	1044: (* Schleppabstand Filter Time ***********************************************************************)	
		getValue(IDxGrp:= 16#6000,	IDxOffs := 16#13,	LEN := SIZEOF(MaxPosLagFilterTime),	pActValue := ADR(MaxPosLagFilterTime),  pSetValue := ADR(SetMaxPosLagFilterTime) );

	1045: (* Physical unit ***********************************************************************)	
		getValue(IDxGrp:= 16#4000,	IDxOffs := 16#5,	LEN := SIZEOF(PhysicalUnit),	pActValue := ADR(PhysicalUnit),  pSetValue := ADR(PhysicalUnit) );
		IF PhysicalUnit[0] = 176 THEN PhysicalUnit := '°'; END_IF		
		
	1046: (*  Drive type ***********************************************************************)	
		getValue(IDxGrp:= 16#7000,	IDxOffs := 16#3,	LEN := SIZEOF(DriveType),	pActValue := ADR(DriveType),  pSetValue := 0 );
			
	ELSE
		state												:= 1;
	END_CASE

(*********************************************************************************************)
END_METHOD

METHOD PROTECTED seqWrite : BOOL //Return value = TRUE if execution finished 
VAR_IN_OUT
	State							:	INT;
END_VAR
(* Write axis parameter ********************************************************************)
	CASE state OF
	1..99: //Wite application spec parameter 
		seqWrite											:= TRUE;
		
	1001: (* Endlagenlimit pos.beschreiben ********************************************************)
		setValue(IDxGrp:= 16#5000,	IDxOffs := 16#E,	LEN := SIZEOF(SetLimitPos),		pActValue := ADR(LimitPos),		pSetValue := ADR(SetLimitPos));

	1002: (* Endlagenlimit neg.beschreiben ********************************************************)
		setValue(IDxGrp:= 16#5000,	IDxOffs := 16#D,	LEN := SIZEOF(SetLimitNeg),		pActValue := ADR(LimitNeg),		pSetValue := ADR(SetLimitNeg));

	1003: (* Endlagenlimit pos. aktiv ****************************************************************)
		IF NOT (SetLimitPosActive XOR LimitPosActive)
			AND NOT WriteAdsPara.BUSY
		THEN 
			state 											:= state + 1;
		ELSE
			_UINT											:= TO_UINT(SetLimitPosActive);
			LimitPosActive									:= SetLimitPosActive;
			setValue(IDxGrp:= 16#5000,	IDxOffs := 16#C,	LEN := SIZEOF(_UINT),		pActValue := 0,		pSetValue := ADR(_UINT));
		END_IF
		
	1004: (* Endlagenlimit neg.aktiv *****************************************************************)
		IF NOT (SetLimitNegActive XOR LimitNegActive) 
			AND NOT WriteAdsPara.BUSY
		THEN 
			state 											:= state + 1;
		ELSE
			_UINT											:= TO_UINT(SetLimitNegActive);
			LimitNegActive									:= SetLimitNegActive; 
			setValue(IDxGrp:= 16#5000,	IDxOffs := 16#B,	LEN := SIZEOF(_UINT),		pActValue := 0,		pSetValue := ADR(_UINT));
		END_IF

	1005: (* Zielfenster setzen **********************************************************************)
		setValue(IDxGrp:= 16#4000,	IDxOffs := 16#16,	LEN := SIZEOF(SetTargetPosWindow),		pActValue := ADR(TargetPosWindow),		pSetValue := ADR(SetTargetPosWindow));

	1006: (* Positionsfenster setzen *****************************************************************)
		setValue(IDxGrp:= 16#4000,	IDxOffs := 16#10,	LEN := SIZEOF(SetPosRangeWindow),		pActValue := ADR(PosRangeWindow),	pSetValue := ADR(SetPosRangeWindow));
		
	1007: (* Bezugsgeschwindigkeit setzen ********************************************************)
		IF AxisType = 2
		THEN 
			state 											:= state +1;
		ELSE
			setValue(IDxGrp:= 16#7000,	IDxOffs := 16#101,	LEN := SIZEOF(SetDynamicsRefVelocity),pActValue := ADR(DynamicsRefVelocity),	pSetValue := ADR(SetDynamicsRefVelocity));
		END_IF


	1008: (* Max.Geschwindigkeit setzen ************************************************************)
		IF AxisType = 2 
		THEN 
			state 											:= state +1;
		ELSE
			setValue(IDxGrp:= 16#4000,	IDxOffs := 16#27,	LEN := SIZEOF(SetDynamicsMaxVelocity),pActValue := ADR(DynamicsMaxVelocity),	pSetValue := ADR(SetDynamicsMaxVelocity));
		END_IF

	1009: (* G0 Geschwindigkeit setzen ****************************************************************)
		setValue(IDxGrp:= 16#4000,	IDxOffs := 16#A,	LEN := SIZEOF(SetG0Velocity),	pActValue := ADR(G0Velocity),	pSetValue := ADR(SetG0Velocity));

	1010: (* Ref.Geschwindigkeit fast setzen *******************************************************)
		setValue(IDxGrp:= 16#4000,	IDxOffs := 16#6,	LEN := SIZEOF(SetRefVelocityPos),	pActValue := ADR(RefVelocityPos),	pSetValue := ADR(SetRefVelocityPos));

	1011: (* Ref.Geschwindigkeit slow setzen *****************************************************)
		setValue(IDxGrp:= 16#4000,	IDxOffs := 16#7,	LEN := SIZEOF(SetRefVelocityNeg),	pActValue := ADR(RefVelocityNeg),	pSetValue := ADR(SetRefVelocityNeg));

	1012: (* Man.Geschwindigkeit fast setzen ******************************************************)
		setValue(IDxGrp:= 16#4000,	IDxOffs := 16#9,	LEN := SIZEOF(SetManVelocityFast),	pActValue := ADR(ManVelocityFast),	pSetValue := ADR(SetManVelocityFast));
		

	1013: (* Man.Geschwindigkeit slow setzen ******************************************************)
		setValue(IDxGrp:= 16#4000,	IDxOffs := 16#8,	LEN := SIZEOF(SetManVelocitySlow),	pActValue := ADR(ManVelocitySlow),	pSetValue := ADR(SetManVelocitySlow));

	1014: (* Kv setzen **************************************************************************************)
		IF AxisType = 2 
		THEN 
			state 											:= state +1;
		ELSE
			setValue(IDxGrp:= 16#6000,	IDxOffs := 16#102,	LEN := SIZEOF(SetKv),pActValue := ADR(Kv),	pSetValue := ADR(SetKv));
		END_IF

	1015: (* Ruck setzen ***********************************************************************************)
		IF AxisType = 2 
		THEN 
			state 											:= state +1;
		ELSE
			setValue(IDxGrp:= 16#4000,	IDxOffs := 16#103,	LEN := SIZEOF(SetJerk),pActValue := ADR(Jerk),	pSetValue := ADR(SetJerk));
		END_IF

	1016: (* Beschleunigung setzen **********************************************************************)
		IF AxisType = 2 
		THEN 
			state 											:= state +1;
		ELSE
			setValue(IDxGrp:= 16#4000,	IDxOffs := 16#101,	LEN := SIZEOF(SetAcc), pActValue := ADR(Acc),	pSetValue := ADR(SetAcc));
		END_IF
	
	1017: (* Verzoegerung setzen ************************************************************************)
		IF AxisType = 2 
		THEN 
			state 											:= state +1;
		ELSE
			setValue(IDxGrp:= 16#4000,	IDxOffs := 16#102,	LEN := SIZEOF(SetDec), pActValue := ADR(Dec),	pSetValue := ADR(SetDec));
		END_IF
		
	1018: (* Schleppabstand setzen **********************************************************************)
		setValue(IDxGrp:= 16#6000,	IDxOffs := 16#12,	LEN := SIZEOF(SetMaxPosLagValue),	pActValue := ADR(MaxPosLagValue),	pSetValue := ADR(SetMaxPosLagValue));

	1019: (* Reserverd *****************************************************************************)
		// Set scaling replaced by Num and Denum  setValue(IDxGrp:= 16#5000,	IDxOffs := 16#6,	LEN := SIZEOF(SetEncScaling),	pActValue := ADR(EncScaling),	pSetValue := ADR(SetEncScaling));
		state 												:= state +1 ;
		
	1020: (* Positions Offset setzen ****************************************************************)
		setValue(IDxGrp:= 16#5000,	IDxOffs := 16#7,	LEN := SIZEOF(SetPosBias),	pActValue := ADR(PosBias),	pSetValue := ADR(SetPosBias));
		
	1021: (* Referenzposition setzen ***************************************************************)
		IF EncType <> 2  AND EncType <> 5 AND EncType <> 7 AND EncType <> 11  AND EncType <> 12 
		THEN
			setValue(IDxGrp:= 16#5000,	IDxOffs := 16#103,	LEN := SIZEOF(SetCalibrationValue),	pActValue := ADR(CalibrationValue),	pSetValue := ADR(SetCalibrationValue));
		ELSE
			state 											:= state +1 ;
		END_IF

	1022: (* Bremsweg positiv **********************************************************************)
		IF AxisType = 2 
		THEN 
			state 											:= state +1;
		ELSE
			setValue(IDxGrp:= 16#4000,	IDxOffs := 16#303,	LEN := SIZEOF(SetBreakingDistancePos), pActValue := ADR(BreakingDistancePos),	pSetValue := ADR(SetBreakingDistancePos));
		END_IF

	1023: (* Bremsweg negativ *********************************************************************)
		IF AxisType = 2
		THEN 
			state 											:= state +1;
		ELSE
			setValue(IDxGrp:= 16#4000,	IDxOffs := 16#304,	LEN := SIZEOF(SetBreakingDistanceNeg), pActValue := ADR(BreakingDistanceNeg),	pSetValue := ADR(SetBreakingDistanceNeg));
		END_IF

	1024: (* Schleppueberwachung ****************************************************************************)
		IF SetMaxPosLagMonitoring = MaxPosLagMonitoring AND NOT WriteAdsPara.BUSY
		THEN 
			state 											:= state +1;
		ELSE
			_UINT											:= TO_UINT(SetMaxPosLagMonitoring);
			MaxPosLagMonitoring								:= SetMaxPosLagMonitoring;					
			setValue(IDxGrp:= 16#6000,	IDxOffs := 16#10,	LEN := SIZEOF(_UINT),	pActValue := 0,	pSetValue := ADR(_UINT));
		END_IF

	1025: (* Referenzierflag ****************************************************************************)
		IF RefFlag = SetRefFlag AND NOT WriteAdsPara.BUSY
		THEN 
			state 											:= state +1;
		ELSE
			_UINT											:= TO_UINT(SetRefFlag);
			RefFlag											:= SetRefFlag;
			setValue(IDxGrp:= 16#5100,	IDxOffs := 16#9,	LEN := SIZEOF(_UINT), pActValue := 0,	pSetValue := ADR(_UINT));
		END_IF
		
	1026: (* PosfensterAktiv ****************************************************************************)
		IF SetPosRangeWindowMonitoring = PosRangeWindowMonitoring AND NOT WriteAdsPara.BUSY
		THEN 
			state 											:= state +1;
		ELSE
			_UINT											:= TO_UINT(SetPosRangeWindowMonitoring);
			PosRangeWindowMonitoring						:= SetPosRangeWindowMonitoring;
			setValue(IDxGrp:= 16#4000,	IDxOffs := 16#F,	LEN := SIZEOF(_UINT), pActValue := 0,	pSetValue := ADR(_UINT));
		END_IF

	1027: (* ZielfensterAktiv ****************************************************************************)
		IF SetTargetPosWindowMonitoring = TargetPosWindowMonitoring AND NOT WriteAdsPara.BUSY
		THEN 
			state 											:= state +1;
		ELSE
			_UINT											:= TO_UINT(SetTargetPosWindowMonitoring);
			TargetPosWindowMonitoring						:= SetTargetPosWindowMonitoring;
			setValue(IDxGrp:= 16#4000,	IDxOffs := 16#15,	LEN := SIZEOF(_UINT), pActValue := 0,	pSetValue := ADR(_UINT));
		END_IF

	1028: (* Modulofaktor ****************************************************************************)
		setValue(IDxGrp:= 16#5000,	IDxOffs := 16#9,	LEN := SIZEOF(SetModuloFactor), pActValue := ADR(ModuloFactor),	pSetValue := ADR(SetModuloFactor));
		
	1029: (* Enc. Zaehlrichtung ****************************************************************************)
		IF SetInvertEncCoutingDir = InvertEncCoutingDir AND NOT WriteAdsPara.BUSY
		THEN 
			state 											:= state +1;
		ELSE
			_UINT											:= TO_UINT(SetInvertEncCoutingDir);
			InvertEncCoutingDir								:= SetInvertEncCoutingDir;
			setValue(IDxGrp:= 16#5000,	IDxOffs := 16#8,	LEN := SIZEOF(_UINT), pActValue := 0,	pSetValue := ADR(_UINT));
		END_IF

	1030: (* Drive  ****************************************************************************)
		IF SetInvertMotorPolarity = InvertMotorPolarity AND NOT WriteAdsPara.BUSY
		THEN 
			state 											:= state +1;
		ELSE
			_UINT											:= TO_UINT(SetInvertMotorPolarity);
			InvertMotorPolarity								:= SetInvertMotorPolarity;
			setValue(IDxGrp:= 16#7000,	IDxOffs := 16#6,	LEN := SIZEOF(_UINT), pActValue := 0,	pSetValue := ADR(_UINT));
		END_IF
		
		
	1031: (* Enc. Modulo start tolerance ****************************************************************************)
		setValue(IDxGrp:= 16#5000,	IDxOffs := 16#1B,	LEN := SIZEOF(SetToleranceWindowModuloStart), pActValue := ADR(ToleranceWindowModuloStart),	pSetValue := ADR(SetToleranceWindowModuloStart));

	1032: (* Set calibration cam search direction inverted ***************************************************************)
		IF SetCalibrInvertDirForCamSearch = CalibrInvertDirForCamSearch	AND NOT WriteAdsPara.BUSY
			OR_ELSE(EncType = 2  OR EncType = 5 OR EncType = 7 OR EncType = 11  OR EncType = 12)
		THEN 
			state 											:= state +1;
		ELSE
			_UINT											:= TO_UINT(SetCalibrInvertDirForCamSearch);
			CalibrInvertDirForCamSearch						:= SetCalibrInvertDirForCamSearch;
			setValue(IDxGrp:= 16#5000,	IDxOffs := 16#101,	LEN := SIZEOF(_UINT), pActValue := 0,	pSetValue := ADR(_UINT));
		END_IF

	1033: (* Set calibration impuls search direction inverted ***************************************************************)
		IF SetCalibrInvertDirForSyncImpSearch = CalibrInvertDirForSyncImpSearch AND NOT WriteAdsPara.BUSY
			OR_ELSE(EncType = 2  OR EncType = 5 OR EncType = 7 OR EncType = 11  OR EncType = 12)
		THEN 
			state 											:= state +1;
		ELSE
			_UINT											:= TO_UINT(SetCalibrInvertDirForSyncImpSearch);
			CalibrInvertDirForSyncImpSearch					:= SetCalibrInvertDirForSyncImpSearch;
			setValue(IDxGrp:= 16#5000,	IDxOffs := 16#102,	LEN := SIZEOF(_UINT), pActValue := 0,	pSetValue := ADR(_UINT));
		END_IF
		
	1034: (* Set calibration mode ***************************************************************)
		IF SetCalibrationMode = CalibrationMode  AND NOT WriteAdsPara.BUSY
			OR_ELSE(EncType = 2  OR EncType = 5 OR EncType = 7 OR EncType = 11  OR EncType = 12)
		THEN 
			state 											:= state +1;		
		ELSE
			setValue(IDxGrp:= 16#5000,	IDxOffs := 16#107,	LEN := SIZEOF(SetCalibrationMode), pActValue := ADR(CalibrationMode),	pSetValue := ADR(SetCalibrationMode));
		END_IF

	1035: (* Scaling numerator **************************************)
		setValue(IDxGrp:= 16#5000,	IDxOffs := 16#23,	LEN := SIZEOF(SetEncScalingNumerator),	pActValue := ADR(EncScalingNumerator),  pSetValue := ADR(SetEncScalingNumerator) );	
			
	1036: (* Scaling denumerator **************************************)
		setValue(IDxGrp:= 16#5000,	IDxOffs := 16#24,	LEN := SIZEOF(SetEncScalingDenominator),	pActValue := ADR(EncScalingDenominator),  pSetValue := ADR(SetEncScalingDenominator) );
		
		//Calculate Act Scaling 
		IF NOT Error THEN  EncScaling	:= EncScalingNumerator / EncScalingDenominator; END_IF
		
	1037: (* Reference system **************************************)
		setValue(IDxGrp:= 16#5000,	IDxOffs := 16#19,	LEN := SIZEOF(SetReferenceSystem),	pActValue := ADR(ReferenceSystem),  pSetValue := ADR(SetReferenceSystem) );	
	
	1038: (* Schleppueberwachung Zeit ****************************************************************************)
		setValue(IDxGrp:= 16#6000,	IDxOffs := 16#13,	LEN := SIZEOF(SetMaxPosLagFilterTime),	pActValue := ADR(MaxPosLagFilterTime),	pSetValue := ADR(SetMaxPosLagFilterTime));
	
	ELSE
		state 												:= 1 ;
	END_CASE
	
(***********************************************************************************************)
END_METHOD

METHOD PROTECTED setValue : BOOL //Return value = TRUE if execution finished and state incremented 
VAR_INPUT
	IDxGrp						:	UDINT;
	IDxOffs						:	UDINT;
	Len							:	UDINT;
	pActValue					:	PVOID; //Address of variable for actual value, can be zero if no corresponding acual value variable exists
	pSetValue					:	PVOID; //Address of variable for set value variable
END_VAR

IF pActValue <> 0 AND pSetValue <> 0 AND_THEN MEMCMP(pSetValue, pActValue, Len) = 0
THEN //Skip write parameter if set and actual value are equel
	state													:= state + 1;	
	setValue												:= TRUE;
ELSE
	WriteAdsPara( Write := TRUE, IdxGrp :=IDxGrp+AxisId, IdxOffs:=IDxOffs, LEN:=Len, SrcAddr:=pSetValue );
	IF NOT WriteAdsPara.BUSY
	THEN
		IF NOT WriteAdsPara.ERR
		THEN
			IF pActValue <> 0 THEN MEMCPY(pActValue, pSetValue, Len); END_IF	
			state											:= state + 1;
		ELSE
			Busy											:= FALSE;
			Error											:= TRUE;
			ErrorId											:= WriteAdsPara.ERRID;
			ErrorText										:= CONCAT('Error write parameter in state:' , TO_STRING(state * -1));
			ErrorText										:= CONCAT(ErrorText , ' Id:');
			ErrorText										:= CONCAT(ErrorText , TO_STRING(ErrorId));
			State											:= 9999;
		END_IF
		WriteAdsPara (Write := FALSE);
		setValue											:= TRUE;
	END_IF		
END_IF
END_METHOD

END_FUNCTION_BLOCK

// POUs/Motion/TF50xx-NC/00_Base/I_AxNcPTP
INTERFACE I_AxNcPTP EXTENDS I_AxNcBase

{attribute 'monitoring' := 'call'}
PROPERTY rMotion : REFERENCE TO AxMotion
GET
END_GET
END_PROPERTY

END_INTERFACE

// POUs/Motion/TF50xx-NC/01_Main/AxMotion
{attribute 'no_check'}
//Nc-axis motion control - start/stop axis  
//based on Tc2_MC2 library
FUNCTION_BLOCK AxMotion EXTENDS AxFbBase
VAR_OUTPUT CONSTANT
	FNC_HALT												:	INT := 0;
	FNC_STOP												:	INT := 1;
	FNC_MOVE_JOG											:	INT := 2;
	FNC_MOVE_ABS											:	INT := 3;
	FNC_MOVE_REL											:	INT := 4;
	FNC_MOVE_ADD											:	INT := 5;
	FNC_MOVE_MOD											:	INT := 6;
	FNC_MOVE_VELO											:	INT := 7;
END_VAR
VAR_INPUT
	Fnc														:	INT (FNC_HALT..FNC_MOVE_VELO) := FNC_HALT;
	JogFwd													:	BOOL := FALSE;
	JogBwd													:	BOOL	:= FALSE;
	BufferMode												:	MC_BufferMode := MC_Aborting;(* 	MC_Aborting,
																											MC_Buffered,
																											MC_BlendingLow,
																											MC_BlendingPrevious,
																											MC_BlendingNext,
																											MC_BlendingHigh *)
	Direction												:	MC_Direction := MC_POSITIVE_DIRECTION;	(*	MC_POSITIVE_DIRECTION,
																														   MC_SHORTeSTATE.WAY,
																														   MC_NEGATIVE_DIRECTION,
																														   MC_CURRENT_DIRECTION *)
	JogMode													:	E_JogMode := MC_JOGMODE_STANDARD_SLOW;	(*	MC_JOGMODE_STANDARD_SLOW
																															MC_JOGMODE_STANDARD_FAST
																															MC_JOGMODE_CONTINOUS
																															MC_JOGMODE_INCHING 
																															MC_JOGeMODE.INCHING_MODULO *)
	Target													:	LREAL; (* Zielposition *)
	Velo														: 	LREAL; (* Zielgeschwindigkeit *)
	Jerk														:	LREAL := 0.0 ; (* Bei 0 werden wird der Ruck aus dem TCManager uebernommen *)
	Acc														:	LREAL := 0.0; (* Bei 0 werden wird die Beschleunigung aus dem TCManager uebernommen *)
	Dec														:	LREAL := 0.0; (* Bei 0 werden wird die Verzoegerung aus dem TCManager uebernommen *)
	MoveOptions												:	ST_MoveOptions;
END_VAR                     								
VAR_IN_OUT                  								
END_VAR                     								
VAR_OUTPUT                  								
END_VAR
VAR
(* Zwischenspeicher **************************************************************************)
	MemFnc													:	INT := -1;
	MemFncAct												:	INT := -1;
	MCFctTxt												:	STRING(25);
	TrigID													:	INT := 2; (* um mit Trig 1 zu starten *)
	MemBufferMode											:	MC_BufferMode;
	ActSetTarget											:	LREAL;
	ActSetVelo												:	LREAL;
	BusyIntern												:	BOOL;

(* Timer *)

(* Trigger *)
	rtExecuteMethod											:	R_TRIG;

(* Instanzierung der MC Bausteine *******************************************************)
	MC_Halt													: 	MC_Halt;
	MC_Stop													: 	MC_Stop;
	MC_MoveVeloPreTrig										: 	MC_MoveVelocity;
	MC_Jog													: 	MC_Jog;

(* Durch entfernen der Kommentarsymbole koennen noch weitere benötigte MC_Move Varianten
	mit ins Programm genommen werden 
*)
	MC_MoveAbsolute											: 	ARRAY[1..2] OF MC_MoveAbsolute;
	MC_MoveModulo											: 	ARRAY[1..2] OF MC_MoveModulo;
	MC_MoveRelative											: 	ARRAY[1..2] OF MC_MoveRelative;
	MC_MoveAdditive											: 	ARRAY[1..2] OF MC_MoveAdditive; 
	MC_MoveVelocity											: 	ARRAY[1..2] OF MC_MoveVelocity; 

(* Dummy Speicher **********************************************************)
	i														: INT := 0 ;

(* Skalierungsfaktor ermitteln *********************************************
	Skalierungsfaktor von 0.1 eintragen. Istpositon "Anfang" merken.
	Antrieb um einen realen Wert "X" mm verfahren. Differenz der
	momentanen Istposition zur Istposition "Anfang" ermitteln.
	SKalierungsfaktor =		realer Fahrweg 
							---------------------------
							Differenz der Istpositionen
*)
END_VAR

	(* Axis motion control 													*)
	(************************************************************************)

(* Execute ***************************************************************************************)
	rtExecute(CLK := Execute XOR(JogBwd AND NOT JogFwd OR JogFwd AND NOT JogBwd));	
	IF rtExecute.Q AND NOT rtExecuteMethod.Q
	THEN
		MemFnc 												:= SEL(JogBwd OR JogFwd, Fnc, FNC_MOVE_JOG) ;
		Busy												:= TRUE;
		Done												:= FALSE;
		Active												:= FALSE;
		Error												:= FALSE;
		ErrorID												:= 0;
		CmdAborted											:= FALSE;
		ErrorText											:= '';
	END_IF

(* Call Method ***********************************************************************************)
	CASE MemFnc OF
	FNC_STOP												:	Stop(Execute);
	FNC_HALT												:	Halt(Execute);
	FNC_MOVE_JOG											:	MoveJog(Execute);
	FNC_MOVE_ABS											:	MoveAbs(Execute);
	FNC_MOVE_REL											:	MoveRel(Execute);
	FNC_MOVE_ADD											:	MoveAdd(Execute);
	FNC_MOVE_MOD											:	MoveMod(Execute);
	FNC_MOVE_VELO											:	MoveVelo(Execute);
	-1:
		IF NOT rtExecute.CLK
		THEN
			Busy											:= FALSE;
			Done											:= FALSE;
			Error											:= FALSE;
			ErrorID											:= 0;
			Active											:= FALSE;
			CmdAborted										:= FALSE;
			ErrorText										:= '';
		END_IF
	ELSE
		Busy												:= FALSE;
		Done												:= FALSE;
		Active												:= FALSE;
		Error												:= Execute;
		ErrorID												:= E_AdsErr.DEVICE_INVALIDPARM;
		CmdAborted											:= FALSE;
		ErrorText											:= CONCAT('invalid parameter value(s) Fnc no: ' , INT_TO_STRING(MemFnc));
	END_CASE

(*************************************************************************************************)

METHOD PRIVATE _MCIntern : BOOL
VAR_INPUT
END_VAR
(* Internal MC Action											*)
(****************************************************************)

(* Check Pointer **********************************************************************)
IF NOT __ISVALIDREF(rAxis) 
THEN
	Busy													:= NOT Error;
	Error													:= TRUE;
	ErrorId													:= E_AdsErr.DEVICE_INVALIDPARM;
	CmdAborted												:= FALSE;
	Done													:= FALSE;
	Active													:= FALSE;
	ErrorText												:= 'Reference rAxis invalid (0)';
	MemFnc													:= SEL(Execute , -1 ,MemFnc); 
	RETURN;
END_IF

(* flag Execute ***********************************************************************)
	rtExecuteMethod(CLK := Execute OR rtExecute.Q);
	IF rtExecuteMethod.Q 
	THEN
		MC_Stop.Execute										:= FALSE;
		MC_Halt.Execute										:= FALSE;
		MC_MoveVeloPreTrig.Execute							:= FALSE;
		MC_MoveModulo[1].Execute 							:= MC_MoveModulo[2].Execute	:= FALSE;
		MC_MoveAbsolute[1].Execute							:= MC_MoveAbsolute[2].Execute	:= FALSE;
		MC_MoveRelative[1].Execute 							:= MC_MoveRelative[2].Execute := FALSE; 
		MC_MoveAdditive[1].Execute 							:= MC_MoveAdditive[2].Execute := FALSE; 
		MC_MoveVelocity[1].Execute 							:= MC_MoveVelocity[2].Execute := FALSE; 
		BusyIntern											:= FALSE;
		MemFncAct 											:= MemFnc;
	END_IF

(* ctrl programm ******************************************************************************)
	CASE MemFncAct OF
	-1: ; //No Fnc started
	FNC_STOP:
		MC_Stop.Execute										:=	Execute; (* Achse Locked solange Stop noch ansteht *)
		MC_Stop.Deceleration 								:= Dec;
		MC_Stop.Jerk 										:= Jerk;
		MC_Stop.Options 									:= MoveOptions;

	FNC_HALT:
		MC_Halt.Execute										:=	NOT MC_Stop.Busy AND Execute; (* Execute if axis is not locked *)
		MC_Halt.BufferMode									:= BufferMode;
		MC_Halt.Deceleration 								:= Dec;
		MC_Halt.Jerk 										:= Jerk;
		MC_Halt.Options 									:= MoveOptions;
		BusyIntern											:= MC_Stop.Busy;

	FNC_MOVE_JOG:
		IF(Execute OR JogBwd OR JogFwd OR MC_Halt.Busy) (* new cmd or stop last cmd busy *)
			AND NOT rAxis.NcToPlc.StateDWord.2  (* NotMoving *)
			AND NOT MC_Jog.Busy (* not if Mc_Jog running *)
			AND NOT rAxis.NcToPlc.StateDWord.5 (* Protected *) (* not if axis coupled or in NCI group *)
			AND NOT MC_Halt.Error AND NOT MC_Halt.CommandAborted
		THEN
			MC_Halt.Execute									:=	TRUE;
			MC_Halt.BufferMode								:= MC_Aborting;
			MC_Halt.Deceleration 							:= Dec;
			MC_Halt.Jerk 									:= Jerk;
			MC_Halt.Options 								:= MoveOptions;
			BusyIntern										:= TRUE;
		ELSE
			MC_Jog.JogBackwards								:= NOT MC_Stop.Busy AND (JogBwd XOR Execute AND Direction = MC_NEGATIVE_DIRECTION);
			MC_Jog.JogForward								:= NOT MC_Stop.Busy AND (JogFwd XOR Execute AND Direction = MC_POSITIVE_DIRECTION);
			MC_Jog.Mode										:= JogMode;
			MC_Jog.Position 								:= Target;
			MC_Jog.Velocity 								:= Velo;
			MC_Jog.Acceleration 							:= Acc;
			MC_Jog.Deceleration 							:= Dec;
			MC_Jog.Jerk 									:= Jerk;
			MC_Halt.Execute									:=	FALSE;
			BusyIntern										:= MC_Stop.Busy;
		END_IF

	FNC_MOVE_ABS..FNC_MOVE_VELO:
		IF MC_Stop.Busy
			OR rAxis.NcToPlc.StateDWord.29 (* MotionCommandsLocked *)
		//	OR MC_Jog.Busy Allow new command even jog is still active
		THEN (* Solange hier rein bis Achse wieder frei und Stop nicht mehr Busy *)
			BusyIntern										:= TRUE;

		ELSIF rAxis.NcToPlc.StateDWord.24 (* CmdBuffered *) 
		THEN (* this section is for aborting a buffered running axis *)
			IF NOT MC_MoveVeloPreTrig.Execute
				AND BufferMode = MC_Aborting
				AND(
				rtExecuteMethod.Q (* new cmd with MC_Aborting to break up current and buffered cmd *)
				OR 		(* or break up current and buffered cmd with new targetpos. *)
				Execute
				AND (Busy OR Done OR CmdAborted) (* dont restart if error is active *)
				AND (ActSetTarget <> Target))
			THEN
				TrigID 										:= 0;
				MC_MoveVeloPreTrig.Execute 					:= TRUE;
				MC_MoveVeloPreTrig.BufferMode 				:= MC_Aborting;
				MC_MoveVeloPreTrig.Velocity 				:= Velo;
				IF rAxis.NcToPlc.StateDWord.10 (* NegativeDirection *) 
				THEN
					MC_MoveVeloPreTrig.Direction 			:= MC_NEGATIVE_DIRECTION;
				ELSE
					MC_MoveVeloPreTrig.Direction 			:= MC_POSITIVE_DIRECTION;
				END_IF
				BusyIntern									:= TRUE;
			ELSE
				;
			END_IF

		ELSE (* ready for start/restart (MC_MoveVeloPreTrig is active) *)
			IF rtExecuteMethod.Q (* new cmd *)
				OR TrigID = 0 (* new cmd with Buffermode aborted *)
				OR(	Execute
				AND (Busy OR Done OR CmdAborted) (* dont restart if error is active *)
				AND (ActSetTarget <> Target OR ActSetVelo <> Velo AND BufferMode = MC_Aborting)) (* restart only with new velo if bufferMode = Aborting *)
			THEN (* new cmd *)
				(* Cancel MoveVeloPreTrig block *)
				IF TrigID = 0 THEN
					MemBufferMode 							:= MC_Aborting;
				ELSE
					MemBufferMode						 	:= BufferMode;
				END_IF

				(* change TrigID *)
				IF TrigID <> 1 THEN
					TrigID 									:= 1;
				ELSE
					TrigID 									:= 2;
				END_IF

				(* Save Act. target and velo *)
				ActSetTarget 								:= Target;
				ActSetVelo 									:= Velo;

				(* Init MC-Blocks *)
				MC_MoveModulo[1].Execute 					:= MC_MoveModulo[2].Execute	:= FALSE;
				MC_MoveAbsolute[1].Execute					:= MC_MoveAbsolute[2].Execute	:= FALSE;
				MC_MoveRelative[1].Execute 					:= MC_MoveRelative[2].Execute := FALSE; 
				MC_MoveAdditive[1].Execute 					:= MC_MoveAdditive[2].Execute := FALSE; 
				MC_MoveVelocity[1].Execute 					:= MC_MoveVelocity[2].Execute := FALSE; 
			END_IF

			CASE MemFncAct OF
			FNC_MOVE_ABS:(* Absolute *);
				MC_MoveAbsolute[TrigID].Execute				:= Execute OR BusyIntern;
				MC_MoveAbsolute[TrigID].BufferMode 			:= MemBufferMode;
				MC_MoveAbsolute[TrigID].Position 			:= Target;
				MC_MoveAbsolute[TrigID].Velocity 			:= Velo;
				MC_MoveAbsolute[TrigID].Acceleration 		:= Acc;
				MC_MoveAbsolute[TrigID].Deceleration 		:= Dec;
				MC_MoveAbsolute[TrigID].Jerk 				:= Jerk;
				MC_MoveAbsolute[TrigID].Options 			:= MoveOptions;

			FNC_MOVE_MOD:(* Modulo *);
				MC_MoveModulo[TrigID].Execute				:= Execute OR BusyIntern;
				MC_MoveModulo[TrigID].BufferMode 			:= MemBufferMode;
				MC_MoveModulo[TrigID].Position 				:= Target;
				MC_MoveModulo[TrigID].Direction 			:= Direction;
				MC_MoveModulo[TrigID].Velocity 				:= Velo;
				MC_MoveModulo[TrigID].Acceleration 			:= Acc;
				MC_MoveModulo[TrigID].Deceleration 			:= Dec;
				MC_MoveModulo[TrigID].Jerk 					:= Jerk;
				MC_MoveModulo[TrigID].Options 				:= MoveOptions;
			
			FNC_MOVE_REL: (* Relativ *)
				MC_MoveRelative[TrigID].Execute				:= Execute OR BusyIntern;
				MC_MoveRelative[TrigID].BufferMode 			:= MemBufferMode;
				MC_MoveRelative[TrigID].Distance 			:= Target;
				MC_MoveRelative[TrigID].Velocity 			:= Velo;
				MC_MoveRelative[TrigID].Acceleration 		:= Acc;
				MC_MoveRelative[TrigID].Deceleration	 	:= Dec;
				MC_MoveRelative[TrigID].Jerk 				:= Jerk;
				MC_MoveRelative[TrigID].Options 			:= MoveOptions;
		
			FNC_MOVE_ADD:(* Rel.Additive *);
				MC_MoveAdditive[TrigID].Execute				:= Execute OR BusyIntern;
				MC_MoveAdditive[TrigID].BufferMode 			:= MemBufferMode;
				MC_MoveAdditive[TrigID].Distance 			:= Target;
				MC_MoveAdditive[TrigID].Velocity 			:= Velo;
				MC_MoveAdditive[TrigID].Acceleration	 	:= Acc;
				MC_MoveAdditive[TrigID].Deceleration	 	:= Dec;
				MC_MoveAdditive[TrigID].Jerk 				:= Jerk;
				MC_MoveAdditive[TrigID].Options 			:= MoveOptions;
			
			FNC_MOVE_VELO:(* Velocity *);
				MC_MoveVelocity[TrigID].Execute				:= Execute OR BusyIntern;
				MC_MoveVelocity[TrigID].BufferMode 			:= MemBufferMode;
				MC_MoveVelocity[TrigID].Direction 			:= Direction;
				MC_MoveVelocity[TrigID].Velocity 			:= Velo;
				MC_MoveVelocity[TrigID].Acceleration 		:= Acc;
				MC_MoveVelocity[TrigID].Deceleration 		:= Dec;
				MC_MoveVelocity[TrigID].Jerk 				:= Jerk;
				MC_MoveVelocity[TrigID].Options 			:= MoveOptions;
			
			ELSE
				MC_Halt.Execute								:=	TRUE; // axis locked as long as Stop is set 
				Error										:= TRUE;
				ErrorId										:= E_AdsErr.DEVICE_INVALIDPARM;
				ErrorText									:= CONCAT('invalid parameter value(s) - Fnc no ', INT_TO_STRING(MemFncAct)) ;
			END_CASE

			(* Reset busy intern *)
			MC_MoveVeloPreTrig.Execute 						:= FALSE;
			BusyIntern										:= FALSE;
		END_IF
	ELSE
		MC_Halt.Execute										:=	TRUE; // axis locked as long as Stop is set
		Error												:= TRUE;
		ErrorId												:= E_AdsErr.DEVICE_INVALIDPARM;
		ErrorText											:= CONCAT('invalid parameter value(s) - Fnc no ', INT_TO_STRING(MemFncAct)) ;
	END_CASE

(****************************************************************************)
(* Work MC Blocks 															*)
(****************************************************************************)

	(* Halt/Stop *)
	MC_Stop(Axis	:= rAxis);
	MC_Halt(Axis	:= rAxis);

	(* Jog *)
	IF MC_Jog.JogBackwards OR MC_Jog.JogForward OR MC_Jog.Busy
		OR MC_Jog.Done OR MC_Jog.Active
		OR MC_Jog.CommandAborted OR MC_Jog.Error
	THEN
		MC_Jog( Axis :=	rAxis);
		MC_Jog.JogBackwards									:= FALSE;
		MC_Jog.JogForward									:= FALSE;
	END_IF

	(* Positionierungen ********************************************)
	(* MC Move Velo PreTrig 1 *)
	IF MC_MoveVeloPreTrig.Execute OR MC_MoveVeloPreTrig.Busy
		OR MC_MoveVeloPreTrig.InVelocity OR MC_MoveVeloPreTrig.Active
		OR MC_MoveVeloPreTrig.CommandAborted OR MC_MoveVeloPreTrig.Error
	THEN
		MC_MoveVeloPreTrig(Axis	:=	rAxis);
	END_IF

	(* Run MC *)
	IF MC_MoveAbsolute[1].Execute OR MC_MoveAbsolute[1].Busy
		OR MC_MoveAbsolute[1].Done OR MC_MoveAbsolute[1].Active
		OR MC_MoveAbsolute[1].CommandAborted OR MC_MoveAbsolute[1].Error
	THEN
		MC_MoveAbsolute[1]( Axis	:=	rAxis);
	END_IF

	IF MC_MoveModulo[1].Execute OR MC_MoveModulo[1].Busy
		OR MC_MoveModulo[1].Done OR MC_MoveModulo[1].Active
		OR MC_MoveModulo[1].CommandAborted OR MC_MoveModulo[1].Error
	THEN
		MC_MoveModulo[1](Axis	:=	rAxis);
	END_IF
	
	IF MC_MoveRelative[1].Execute OR MC_MoveRelative[1].Busy
		OR MC_MoveRelative[1].Done OR MC_MoveRelative[1].Active
		OR MC_MoveRelative[1].CommandAborted OR MC_MoveRelative[1].Error
	THEN
		MC_MoveRelative[1](Axis	:=	rAxis);
	END_IF
	
	IF MC_MoveAdditive[1].Execute OR MC_MoveAdditive[1].Busy
		OR MC_MoveAdditive[1].Done OR MC_MoveAdditive[1].Active
		OR MC_MoveAdditive[1].CommandAborted OR MC_MoveAdditive[1].Error
	THEN
		MC_MoveAdditive[1](Axis	:=	rAxis);
	END_IF
	
	IF MC_MoveVelocity[1].Execute OR MC_MoveVelocity[1].Busy
		OR MC_MoveVelocity[1].Active OR MC_MoveVelocity[1].InVelocity
		OR MC_MoveVelocity[1].CommandAborted OR MC_MoveVelocity[1].Error
	THEN
		MC_MoveVelocity[1](Axis	:=	rAxis);
	END_IF

	(* MC Move Velo PreTrig 2 **************************************)
	(* Run Trig 2 *)
	IF MC_MoveAbsolute[2].Execute OR MC_MoveAbsolute[2].Busy
		OR MC_MoveAbsolute[2].Done OR MC_MoveAbsolute[2].Active
		OR MC_MoveAbsolute[2].CommandAborted OR MC_MoveAbsolute[2].Error
	THEN
		MC_MoveAbsolute[2](Axis	:=	rAxis);
	END_IF

	IF MC_MoveModulo[2].Execute OR MC_MoveModulo[2].Busy
		OR MC_MoveModulo[2].Done OR MC_MoveModulo[2].Active
		OR MC_MoveModulo[2].CommandAborted OR MC_MoveModulo[2].Error
	THEN
		MC_MoveModulo[2](Axis	:=	rAxis);
	END_IF

	
	IF MC_MoveRelative[2].Execute OR MC_MoveRelative[2].Busy
		OR MC_MoveRelative[2].Done OR MC_MoveRelative[2].Active
		OR MC_MoveRelative[2].CommandAborted OR MC_MoveRelative[2].Error
	THEN
		MC_MoveRelative[2](Axis	:=	rAxis);
	END_IF
	
	IF MC_MoveAdditive[2].Execute OR MC_MoveAdditive[2].Busy
		OR MC_MoveAdditive[2].Done OR MC_MoveAdditive[2].Active
		OR MC_MoveAdditive[2].CommandAborted OR MC_MoveAdditive[2].Error
	THEN
		MC_MoveAdditive[2](Axis	:=	rAxis);
	END_IF

	
	IF MC_MoveVelocity[2].Execute OR MC_MoveVelocity[2].Busy
		OR MC_MoveVelocity[2].Active OR MC_MoveVelocity[2].InVelocity
		OR MC_MoveVelocity[2].CommandAborted OR MC_MoveVelocity[2].Error
	THEN
		MC_MoveVelocity[2](Axis	:=	rAxis);
	END_IF

(******************************************************************************)
(* Ctrl Status 																					*)
(******************************************************************************)
	IF MemFncAct = FNC_STOP
	THEN (* as long as MC_Stop running the axis is locked *)
		MCFctTxt											:= 'MC_STOP';
		Done 												:= MC_Stop.Done;
		Busy 												:= MC_Stop.Busy;
		Active 												:= MC_Stop.Active;
		CmdAborted 											:= MC_Stop.CommandAborted;
		Error												:= MC_Stop.Error;
		ErrorId												:= MC_Stop.ErrorId;
		ErrorText											:= SEL(Error , '' ,  CONCAT('Error MC_STOP id: ',  UDINT_TO_STRING(Errorid)));

	ELSIF MemFncAct = FNC_HALT
	THEN
		MCFctTxt											:= 'MC_HALT';
		Done 												:= MC_Halt.Done;
		Busy 												:= MC_Halt.Busy;
		Active 												:= MC_Halt.Active;
		CmdAborted 	 										:= MC_Halt.CommandAborted;
		Error												:= MC_Halt.Error;
		ErrorId												:= MC_Halt.ErrorId;
		ErrorText											:= SEL(Error , '' ,  CONCAT('Error MC_HALT id: ',  UDINT_TO_STRING(Errorid)));

	ELSIF BusyIntern
	THEN
		MCFctTxt											:= CONCAT('BUSY INTERN at Fnc no: ', INT_TO_STRING(MemFncAct));
		Busy												:= BusyIntern;
		Done 												:= FALSE;
		Active 												:= FALSE;
		CmdAborted 											:= FALSE;
		Error												:=	FALSE;
		ErrorId												:= 0;
		ErrorText											:= '';

	ELSIF MemFncAct = FNC_MOVE_JOG
	THEN
		MCFctTxt											:= 'MC_JOG';
		Done 												:= MC_Jog.Done;
		Busy 												:= MC_Jog.Busy;
		Active 												:= MC_Jog.Active;
		CmdAborted 	 										:= MC_Jog.CommandAborted AND NOT rAxis.NcToPlc.StateDWord.26 AND NOT rAxis.NcToPlc.StateDWord.27  (* Software limit exceeded *) ;
		Error												:= MC_Jog.Error;
		ErrorId												:= MC_Jog.ErrorId;
		ErrorText											:= SEL(Error , '' ,  CONCAT('Error MC_JOG id: ',  UDINT_TO_STRING(Errorid)));

	ELSIF MC_MoveVeloPreTrig.Execute
		OR TrigID = 0
	THEN (* Pretrig Block *)
		MCFctTxt											:= 'MC_MoveVeloPreTrig';
		Done												:= FALSE;
		Busy												:= MC_MoveVeloPreTrig.Busy;
		Active 												:= MC_MoveVeloPreTrig.Active;
		CmdAborted 	 										:= MC_MoveVeloPreTrig.CommandAborted;
		Error												:= MC_MoveVeloPreTrig.Error;
		ErrorId												:= MC_MoveVeloPreTrig.ErrorId;
		ErrorText											:= SEL(Error , '' ,  CONCAT('Error MC_MoveVeloPreTrig id: ',  UDINT_TO_STRING(Errorid)));

	ELSIF MemFncAct = FNC_MOVE_ABS
	THEN (* Absolut *)
		MCFctTxt											:= CONCAT('MC_MoveAbs TrigID No:',INT_TO_STRING(TrigID));
		Done 												:= MC_MoveAbsolute[TrigID].Done;
		Busy 												:= MC_MoveAbsolute[TrigID].Busy;
		Active 												:= MC_MoveAbsolute[TrigID].Active;
		CmdAborted 	 										:= MC_MoveAbsolute[TrigID].CommandAborted;
		Error												:= MC_MoveAbsolute[TrigID].Error;
		ErrorId												:= MC_MoveAbsolute[TrigID].ErrorId;
		ErrorText											:= SEL(Error , '' ,  CONCAT('Error MC_MoveAbsolute id: ',  UDINT_TO_STRING(Errorid)));
	
	ELSIF MemFncAct = FNC_MOVE_MOD
	THEN (* Modulo *)
		MCFctTxt											:= CONCAT('MC_MoveModulo TrigID No:',INT_TO_STRING(TrigID));
		Done 												:= MC_MoveModulo[TrigID].Done;
		Busy 												:= MC_MoveModulo[TrigID].Busy;
		Active 												:= MC_MoveModulo[TrigID].Active;
		CmdAborted 											:= MC_MoveModulo[TrigID].CommandAborted;
		Error												:= MC_MoveModulo[TrigID].Error;
		ErrorId												:= MC_MoveModulo[TrigID].ErrorId;
		ErrorText											:= SEL(Error , '' ,  CONCAT('Error MC_MoveModulo id: ',  UDINT_TO_STRING(Errorid)));

	ELSIF MemFncAct = FNC_MOVE_REL
	THEN (* Relativ *)
		MCFctTxt											:= CONCAT('MC_MoveRelative TrigID No:',INT_TO_STRING(TrigID));
		Done 												:= MC_MoveRelative[TrigID].Done;
		Busy 												:= MC_MoveRelative[TrigID].Busy;
		Active 												:= MC_MoveRelative[TrigID].Active;
		CmdAborted 	 										:= MC_MoveRelative[TrigID].CommandAborted;
		Error												:= MC_MoveRelative[TrigID].Error;
		ErrorId												:= MC_MoveRelative[TrigID].ErrorId;
		ErrorText											:= SEL(Error , '' ,  CONCAT('Error MC_MoveRelative id: ',  UDINT_TO_STRING(Errorid)));

	ELSIF MemFncAct = FNC_MOVE_ADD
	THEN (* Rel.Additive *)
		MCFctTxt											:= CONCAT('MC_MoveAdditive TrigID No:',INT_TO_STRING(TrigID));
		Done 												:= MC_MoveAdditive[TrigID].Done;
		Busy 												:= MC_MoveAdditive[TrigID].Busy;
		Active 												:= MC_MoveAdditive[TrigID].Active;
		CmdAborted 	 										:= MC_MoveAdditive[TrigID].CommandAborted;
		Error												:= MC_MoveAdditive[TrigID].Error;
		ErrorId												:= MC_MoveAdditive[TrigID].ErrorId;
		ErrorText											:= SEL(Error , '' ,  CONCAT('Error MC_MoveAdditive id: ',  UDINT_TO_STRING(Errorid)));
		
	ELSIF MemFncAct = FNC_MOVE_VELO
	THEN (* Velocity *)
		MCFctTxt											:= CONCAT('MC_MoveVelo TrigID No:',INT_TO_STRING(TrigID));
		Active 												:= MC_MoveVelocity[TrigID].Active;
		Busy 												:= MC_MoveVelocity[TrigID].Busy ;
		CmdAborted 	 										:= MC_MoveVelocity[TrigID].CommandAborted;
		Error												:= MC_MoveVelocity[TrigID].Error;
		ErrorId												:= MC_MoveVelocity[TrigID].ErrorId;
		ErrorText											:= SEL(Error , '' ,  CONCAT('Error MC_MoveVelocity id: ',  UDINT_TO_STRING(Errorid)));
		
	ELSIF MemFncAct > 0
	THEN
		MCFctTxt											:= CONCAT('Unknown Fnc no:', INT_TO_STRING(MemFncAct));
	ELSE                    							
		MCFctTxt											:= SEL(BusyIntern, 'NoAction' , 'Busy intern');
		Busy												:= BusyIntern;
		Done 												:= FALSE;
		Active 												:= FALSE;
		CmdAborted 											:= FALSE;
		IF Error THEN LastErrorId := ErrorId; END_IF
		Error												:=	FALSE;
		ErrorId												:= 0;
		ErrorText											:= '';
	END_IF

(* End funcktion *********************************************************************************)
	IF 	NOT rtExecuteMethod.CLK 
		AND NOT Busy 
		AND NOT Error 
		AND NOT Done 
		AND NOT Active 
		AND NOT CmdAborted
	THEN																	
		IF MC_Jog.Busy
			OR MC_Halt.Busy
			OR MC_Stop.Busy
			OR MC_MoveVeloPreTrig.Busy
			OR MC_MoveAbsolute[1].Busy OR MC_MoveAbsolute[2].Busy
			OR MC_MoveModulo[1].Busy OR MC_MoveModulo[2].Busy
			OR MC_MoveRelative[1].Busy OR MC_MoveRelative[2].Busy 
			OR MC_MoveAdditive[1].Busy OR MC_MoveAdditive[2].Busy 
			OR MC_MoveVelocity[1].Busy OR MC_MoveVelocity[2].Busy 
		THEN (* Ablauffehler , es darf kein Baustein an dieser Stelle Busy sein *)
			MemFnc											:= -2;
		ELSE                								
			MemFnc											:= -1;
		END_IF              	
	END_IF
	
(* Return value ***********************************************************************************)
	_MCIntern												:= TRUE;

(**************************************************************************************************)
END_METHOD

METHOD PUBLIC halt : BOOL //Return value = TRUE if busy
//required parameter
//rAxis
//BufferMode
//Dec
//Jerk
//MoveOptions
VAR_INPUT
	Execute													:	BOOL;
END_VAR
MemFnc 														:= FNC_HALT;
THIS^.Execute												:= Execute;
_MCIntern();            									
Halt														:= Busy;
END_METHOD

METHOD PUBLIC jogOff : BOOL //Return value = TRUE if executio finished
VAR_INPUT
END_VAR
JogBwd 														:= JogFwd := FALSE;
IF __ISVALIDREF(rAxis)
THEN
	JogOff 													:= MemFnc = FNC_MOVE_JOG AND NOT rAxis.Status.Moving;
ELSE
	JogOff 													:= MemFnc = FNC_MOVE_JOG;
END_IF
END_METHOD

METHOD PUBLIC moveAbs : BOOL //Return value = TRUE if busy
//required parameter
//rAxis
//BufferMode
//Target
//Velo
//Acc
//Dec
//Jerk
//MoveOptions
VAR_INPUT
	Execute													:	BOOL;
END_VAR
MemFnc 														:= FNC_MOVE_ABS;
THIS^.Execute												:= Execute;
_MCIntern();            									
MoveAbs														:= Busy;
END_METHOD

METHOD PUBLIC moveAdd : BOOL //Return value = TRUE if busy
//required parameter
//rAxis
//BufferMode
//Target
//Velo
//Acc
//Dec
//Jerk
//MoveOptions
VAR_INPUT
	Execute													:	BOOL;
END_VAR
MemFnc 														:= FNC_MOVE_ADD;
THIS^.Execute												:= Execute;
_MCIntern();            									
MoveAdd														:= Busy;
END_METHOD

METHOD PUBLIC moveJog : BOOL  //Return value = TRUE if busy
//required parameter
//rAxis
//Direction
//JogMode	
//Target
//Velo
//Acc
//Dec
//Jerk
VAR_INPUT
	Execute													:	BOOL;
END_VAR
MemFnc 														:= FNC_MOVE_JOG;
THIS^.Execute												:= Execute;
_MCIntern();        										
MoveJog														:= Busy;
END_METHOD

METHOD PUBLIC moveMod : BOOL //Return value = TRUE if busy
//required parameter
//rAxis
//BufferMode
//Target
//Direction
//Velo
//Acc
//Dec
//Jerk
//MoveOptions
VAR_INPUT
	Execute													:	BOOL;
END_VAR
MemFnc 														:= FNC_MOVE_MOD;
THIS^.Execute												:= Execute;
_MCIntern();            									
MoveMod														:= Busy;
END_METHOD

METHOD moveRel : BOOL //Return value = TRUE if busy
//required parameter
//rAxis
//BufferMode
//Target
//Velo
//Acc
//Dec
//Jerk
//MoveOptions
VAR_INPUT
	Execute													:	BOOL;
END_VAR
MemFnc 														:= FNC_MOVE_REL;
THIS^.Execute												:= Execute;
_MCIntern();            									
MoveRel														:= Busy;
END_METHOD

METHOD PUBLIC moveVelo : BOOL //Return value = TRUE if busy
//required parameter
//rAxis
//BufferMode
//Direction
//Velo
//Acc
//Dec
//Jerk
//MoveOptions
VAR_INPUT
	Execute													:	BOOL;
END_VAR
MemFnc														:= FNC_MOVE_VELO;
THIS^.Execute												:= Execute;
_MCIntern();            									
MoveVelo													:= Busy;
END_METHOD

METHOD PUBLIC stop : BOOL //Return value = TRUE if busy
//required parameter
//rAxis
//Dec
//Jerk
//MoveOptions
VAR_INPUT
	Execute													:	BOOL;
END_VAR
MemFnc 														:= FNC_STOP;
THIS^.Execute												:= Execute;
_MCIntern();            									
Stop														:= busy;
END_METHOD

END_FUNCTION_BLOCK

// POUs/Motion/TF50xx-NC/02_Options/Coupling/AxCamming
{attribute 'no_check'}
//Nc-axis camming (cam tabel) control
//based on Tc2_MC2_Camming library
FUNCTION_BLOCK AxCamming EXTENDS AxFbBase
VAR_OUTPUT CONSTANT
	FNC_CAM_OUT												:	INT := 0;
	FNC_CAM_IN												:	INT := 1;
END_VAR                     								
VAR_INPUT                   								
	Fnc														:	INT (FNC_CAM_OUT..FNC_CAM_IN) := FNC_CAM_OUT;
	MasterOffset											:	LREAL		:= 0.0;
	SlaveOffset												:	LREAL 	:= 0.0;
	MasterScaling											:	LREAL 	:= 1.0;
	SlaveScaling											:	LREAL 	:= 1.0;
	MasterScalingMode										:	MC_CamScalingMode := MC_CAMSCALING_USERDEFINED;
	SlaveScalingMode										:	MC_CamScalingMode := MC_CAMSCALING_USERDEFINED;
	StartMode  												:	MC_StartMode := MC_STARTMODE_ABSOLUTE; 	(* StartMode determines whether the cam plate position is interpreted absolute OR relative TO the coupling position.StartMode can be relative OR absolute FOR master (X coordinate) AND slave (Y coordinate). *)
	TableID  												:	MC_CAM_ID; 		(*ID der Kurvenscheibe mit der gekoppelt wird *)
	ActivationMode											:	MC_CamActivationMode := MC_CAMACTIVATION_INSTANTANEOUS;
	ActivationPosition										:	LREAL := 0.0;
	InterpolationType										:	MC_InterpolationType := MC_INTERPOLATIONTYPE_LINEAR;

	rMasterAxis												:	REFERENCE TO AXIS_REF := 0;
END_VAR
VAR_IN_OUT
END_VAR
VAR_OUTPUT
END_VAR
VAR
(* cache *******************************************************************)
	MemFnc													:	INT := -1;

(* timer *)

(* trigger *)

(* MC-function-block instances *********************************************)
	MC_CamIn												:	MC_CamIn;
	MC_CamOut												:	MC_CamOut;

END_VAR

	(* NC axis cam table control														*)
	(************************************************************************************)

(* Execute ***************************************************************************************)
	rtExecute(CLK := Execute);
	IF rtExecute.Q
		AND MemFnc < 0
	THEN
		MemFnc 												:= Fnc ;
		Busy												:= TRUE;
		Done												:= FALSE;
		Error												:= FALSE;
		ErrorID												:= 0;
		CmdAborted											:= FALSE;
		ErrorText											:= '';
	END_IF

(* Call Method ***********************************************************************************)
	CASE MemFnc OF
	FNC_CAM_OUT:
		CamOut(Execute);

	FNC_CAM_IN:
		CamIn(Execute);

	-1:
		IF NOT Execute
		THEN
			Busy											:= FALSE;
			Done											:= FALSE;
			Error											:= FALSE;
			ErrorID											:= 0;
			CmdAborted										:= FALSE;
			ErrorText										:= '';
		END_IF                              				
	ELSE                                    				
		Busy												:= FALSE;
		Done												:= FALSE;
		Error												:= Execute;
		ErrorID												:= E_AdsErr.DEVICE_INVALIDPARM;
		CmdAborted											:= FALSE;
		ErrorText											:= CONCAT('invalid parameter value(s) Fnc no: ' , INT_TO_STRING(MemFnc));
	END_CASE

(*************************************************************************************************)

METHOD PUBLIC camIn : BOOL //Return value = TRUE if busy
//required parameter
//rAxis
//rMasterAxis
//MasterOffset
//SlaveOffset
//MasterScaling
//SlaveScaling
//StartMode
//CamTableID
//Options
VAR_INPUT
	Execute													:	BOOL;
END_VAR
MemFnc														:= FNC_CAM_IN;
THIS^.Execute												:= Execute;
	
IF NOT __ISVALIDREF(rAxis) 
THEN
	Busy													:= NOT Error;
	Error													:= TRUE;
	ErrorId													:= E_AdsErr.DEVICE_INVALIDPARM;
	CmdAborted												:= FALSE;
	Done													:= FALSE;
	Active													:= FALSE;
	ErrorText												:= 'Reference rAxis invalid (0)';
	MemFnc													:= SEL(Execute , -1 ,MemFnc); 
	RETURN;
ELSIF NOT __ISVALIDREF(rMasterAxis)
THEN
	Busy													:= NOT Error;
	Error													:= TRUE;
	ErrorId													:= E_AdsErr.DEVICE_INVALIDPARM;
	CmdAborted												:= FALSE;
	Done													:= FALSE;
	ErrorText												:= 'Reference rMasterAxis invalid (0)';
	MemFnc													:= SEL(Execute , -1 ,MemFnc); 
	RETURN;
END_IF
	MC_CamIn.Options.ActivationMode							:= ActivationMode;
	MC_CamIn.Options.ActivationPosition						:= ActivationPosition;
	MC_CamIn.Options.MasterScalingMode						:= MasterScalingMode;
	MC_CamIn.Options.SlaveScalingMode						:= SlaveScalingMode;
	MC_CamIn.Options.InterpolationType						:= InterpolationType;

	MC_CamIn(
		Execute			:= Execute,
		MasterOffset	:= MasterOffset,
		SlaveOffset		:= SlaveOffset,
		MasterScaling	:= MasterScaling,
		SlaveScaling	:= SlaveScaling,
		StartMode		:= StartMode,
		CamTableID		:= TableID,
		BufferMode		:= ,
		Options			:= ,
		Master			:= rMasterAxis,
		Slave			:= rAxis,
		InSync			=> Done,
		Busy			=> Busy,
		Active			=> Active,
		CommandAborted	=> CmdAborted,
		Error			=> Error,
		ErrorID			=> ErrorID);

	IF Error THEN
		LastErrorId											:= ErrorId;
		ErrorText 											:= CONCAT('MC_CamIn ID:' , UDINT_TO_STRING(ErrorId));
	ELSE                    								
		ErrorText 											:= '';
	END_IF
	IF NOT MC_CamIn.Execute AND NOT Busy
	THEN
		MemFnc												:= -1  ;
	END_IF
END_METHOD

METHOD PUBLIC camOut : BOOL //Return value = TRUE if busy
//required parameter
//rAxis
VAR_INPUT
	Execute													:	BOOL;
END_VAR
	MemFnc													:= FNC_CAM_OUT;
	THIS^.Execute											:= Execute;
	
IF NOT __ISVALIDREF(rAxis) 
THEN
	Busy													:= NOT Error;
	Error													:= TRUE;
	ErrorId													:= E_AdsErr.DEVICE_INVALIDPARM;
	CmdAborted												:= FALSE;
	Done													:= FALSE;
	Active													:= FALSE;
	ErrorText												:= 'Reference rAxis invalid (0)';
	MemFnc													:= SEL(Execute , -1 ,MemFnc); 
	RETURN;
END_IF
	
	MC_CamOut(
		Execute	:= Execute,
		Options	:= ,
		Slave	:= rAxis,
		Done	=> Done,
		Busy	=> Busy,
		Error	=> Error,
		ErrorID	=> ErrorID);

	Active													:= Busy;
	CmdAborted												:= FALSE;

	IF Error THEN
		LastErrorId											:= ErrorId;
		ErrorText 											:= CONCAT('MC_CamOut ID:' , UDINT_TO_STRING(ErrorId));
	ELSE
		ErrorText 											:= '';
	END_IF

	IF NOT Execute AND NOT Busy
	THEN
		MemFnc												:= -1;
	END_IF
END_METHOD

END_FUNCTION_BLOCK

// POUs/Motion/TF50xx-NC/02_Options/Coupling/AxFlyingSaw
{attribute 'no_check'}
//Nc-axis flying saw control
//based on Tc2_MC2_FlyingSaw library
FUNCTION_BLOCK AxFlyingSaw EXTENDS AxFbBase
VAR_OUTPUT CONSTANT
	FNC_GEAR_OUT											:	INT := 0;
	FNC_GEAR_IN_VELO										:	INT := 1;
	FNC_GEAR_IN_POS											:	INT := 2;
END_VAR                     								
VAR_INPUT                   								
	Fnc														:	INT (FNC_GEAR_OUT..FNC_GEAR_IN_POS) := FNC_GEAR_OUT;
	RatioNumerator											:	LREAL := 1.0; (* Getriebefaktor Numerator/Zähler *)
	RatioDenominator										:	UINT := 1; (* Getriebefaktor Denominator/Nenner *)
	MasterSyncPosition										: 	LREAL := 0.0;
	SlaveSyncPosition										: 	LREAL := 0.0;
	MasterStartDistance										: 	LREAL := 0.0;
	SyncMode												: 	ST_SyncMode; (*... mode ...
																						GearInSyncMode : E_GearInSyncMode;
                            								
																					... 32 bit check mask ... 
																						GearInSync_CheckMask_MinPos : BOOL;
																						GearInSync_CheckMask_MaxPos : BOOL;
																						GearInSync_CheckMask_MaxVelo : BOOL;
																						GearInSync_CheckMask_MaxAcc : BOOL;
																						GearInSync_CheckMask_MaxDec : BOOL;
																						GearInSync_CheckMask_MaxJerk : BOOL;
																						GearInSync_CheckMask_OvershootPos : BOOL;
																						GearInSync_CheckMask_UndershootPos : BOOL;
																						GearInSync_CheckMask_OvershootVelo : BOOL;
																						GearInSync_CheckMask_UndershootVelo : BOOL;
																						GearInSync_CheckMask_OvershootVeloZero : BOOL;
																						GearInSync_CheckMask_UndershootVeloZero : BOOL;
																				
																					... operation masks ...
																						GearInSync_OpMask_RollbackLock : BOOL;
																						GearInSync_OpMask_InstantStopOnRollback : BOOL;
																						GearInSync_OpMask_PreferConstVelo : BOOL;
																						GearInSync_OpMask_IgnoreMasterAcc : BOOL;*)
	Velo													:	LREAL := 0.0;	(* Flying Saw ... Max Slave-Geschwindigkeit in Synchronisierungsphase. Bei 0 --> Systemmanager-Daten. Achtung: Geschwindigkeit wird nur überprüft, wenn die Überprüfung mit der Variablen SyncMode aktiviert wird.*)
	Acc														:	LREAL := 0.0; (* Bei 0 werden wird die Beschleunigung aus dem TCManager uebernommen *)
	Dec														:	LREAL := 0.0; (* Bei 0 werden wird die Verzoegerung aus dem TCManager uebernommen *)
	Jerk													:	LREAL := 0.0; (* Bei 0 werden wird der Ruck aus dem TCManager uebernommen *)
(*	BufferMode												:	MC_BufferMode := MC_Aborting;(* 	MC_Aborting,
																												MC_Buffered,
																												MC_BlendingLow,
																												MC_BlendingPrevious,
																												MC_BlendingNext,
																												MC_BlendingHigh *)
*)                          								
(*	Options 												: 	ST_MOVEOptions; *)
//	rCamTableCharac 										:  REFERENCE TO MC_FlyingSawCharacValues; (* Struktur mit den charakteristischen Kennwerten.*)
	rMasterAxis												:	REFERENCE TO AXIS_REF := 0;
END_VAR                     								
VAR_IN_OUT                  								
END_VAR                     								
VAR_OUTPUT                  								
	StartSync 												:  BOOL;  (* Flying Saw*)
END_VAR
VAR
(* cache **************************************************************************)
	MemFnc													:	INT := -1;
                            								
(* timer *)                 								
                            	
(* trigger *)               	
                            	
(* MC-function-block instances *****************************************************)
	MC_GearOut												:	MC_GearOut;
	MC_GearInVelo 											:  MC_GearInVelo;
	MC_GearInPos											:  MC_GearInPos;	
//	MC_ReadCharacteristics									:  MC_ReadFlyingSawCharacteristics; (* charakteristischen Kennwerte der Synchronisierungsphase ausgelesen *)

(* Dummy storage *******************************************************************)
(*	i,j		: INT := 0 ; *)
	Dummy 	: BOOL; 
END_VAR

	(************************************************************************************)
	(*																					*)
	(*		B E C K H O F F   N E W   A U T O M A T I O N   T E C H N O L O G Y    		*)
	(*																					*)
	(*		Eiserstr.5	D-33415 Verl	Germany	phone:	+49-5246-0	www.Beckhoff.Com	*)
    (*																					*)
    (*		Bausteinbeschreibung	:	Flying Saw Achs Baustein						*)
	(*		TwinCAT-Version			:	3.x or higher									*)
	(*		Version					:	V3.0 / 03/13									*)
	(*		Lib						:	TcMC2_FlyingSaw.lib 							*)
 	(*		Autor					:	DS												*)
	(*																					*)
	(************************************************************************************)

(* Execute ***************************************************************************************)
	rtExecute(CLK := Execute);
	IF rtExecute.Q
		AND MemFnc < 0
	THEN
		MemFnc 												:= Fnc ;
		Busy												:= TRUE;
		Done												:= FALSE;
		Error												:= FALSE;
		ErrorID												:= 0;
		CmdAborted											:= FALSE;
		ErrorText											:= '';
	END_IF

(* Call Method ***********************************************************************************)
	CASE MemFnc OF
	FNC_GEAR_OUT:
		GearOut(Execute);

	FNC_GEAR_IN_VELO:
		GearInVelo(Execute);

	FNC_GEAR_IN_POS:
		GearInPos(Execute);

	-1:
		IF NOT Execute
		THEN
			StartSync										:= FALSE;
			Busy											:= FALSE;
			Done											:= FALSE;
			Error											:= FALSE;
			ErrorID											:= 0;
			CmdAborted										:= FALSE;
			ErrorText										:= '';
		END_IF                          					
	ELSE                                					
		StartSync											:= FALSE;
		Busy												:= FALSE;
		Done												:= FALSE;
		Error												:= Execute;
		ErrorID												:= E_AdsErr.DEVICE_INVALIDPARM;
		CmdAborted											:= FALSE;
		ErrorText											:= CONCAT('invalid parameter value(s) Fnc no: ' , INT_TO_STRING(MemFnc));
	END_CASE

(*************************************************************************************************)

METHOD PUBLIC gearInPos : BOOL //Return value = TRUE if busy
//required parameter
//rAxis
//rMasterAxis
//RatioNumerator
//RatioDenominator
//MasterSyncPosition
//SlaveSyncPosition
//SyncMode
//MasterStartDistance
//Velo
//Acc
//Dec
//Jerk
VAR_INPUT
	Execute													:	BOOL;
END_VAR
MemFnc														:= FNC_GEAR_IN_POS;
THIS^.Execute												:= Execute;
	
IF NOT __ISVALIDREF(rAxis) 
THEN
	Busy													:= NOT Error;
	Error													:= TRUE;
	ErrorId													:= E_AdsErr.DEVICE_INVALIDPARM;
	CmdAborted												:= FALSE;
	Done													:= FALSE;
	Active													:= FALSE;
	ErrorText												:= 'Reference rAxis invalid (0)';
	MemFnc													:= SEL(Execute , -1 ,MemFnc); 
	RETURN;
ELSIF NOT __ISVALIDREF(rMasterAxis)
THEN
	Busy													:= NOT Error;
	Error													:= TRUE;
	ErrorId													:= E_AdsErr.DEVICE_INVALIDPARM;
	CmdAborted												:= FALSE;
	Done													:= FALSE;
	ErrorText												:= 'Reference rMasterAxis invalid (0)';
	MemFnc													:= SEL(Execute , -1 ,MemFnc); 
	RETURN;
END_IF

	MC_GearInPos(
		Execute				:= Execute,
		RatioNumerator		:= RatioNumerator,
		RatioDenominator	:= RatioDenominator,
		MasterSyncPosition	:= MasterSyncPosition,
		SlaveSyncPosition	:= SlaveSyncPosition,
		SyncMode			:= SyncMode,
		MasterStartDistance	:= MasterStartDistance,
		Velocity			:= Velo,
		Acceleration		:= Acc,
		Deceleration		:= Dec,
		Jerk				:= Jerk,
		BufferMode			:= ,
		Options				:= ,
		Master				:= rMasterAxis,
		Slave				:= rAxis,
		StartSync			=> StartSync,
		InSync				=> Done,
		Busy				=> Busy,
		Active				=> Active,
		CommandAborted		=> CmdAborted,
		Error				=> Error,
		ErrorID				=> ErrorID);
		
	

	IF Error THEN
		LastErrorId											:= ErrorId;
		ErrorText 											:= CONCAT('MC_GearInPos ID:' , UDINT_TO_STRING(ErrorId));
	ELSE
		ErrorText 											:= '';
	END_IF

	IF NOT Execute AND NOT Busy
	THEN
		MemFnc												:= -1;
	END_IF
	
	GearInPos												:= Busy;
END_METHOD

METHOD PUBLIC gearInVelo : BOOL //Return value = TRUE if busy
//required parameter
//rAxis
//rMasterAxis
//RatioNumerator
//RatioDenominator
//SyncMode
//Velo
//Acc
//Dec
//Jerk
VAR_INPUT
	Execute													:	BOOL;
END_VAR
MemFnc														:= FNC_GEAR_IN_VELO;
THIS^.Execute												:= Execute;
	
IF NOT __ISVALIDREF(rAxis)
THEN
	Busy													:= NOT Error;
	Error													:= TRUE;
	ErrorId													:= E_AdsErr.DEVICE_INVALIDPARM;
	CmdAborted												:= FALSE;
	Done													:= FALSE;
	Active													:= FALSE;
	ErrorText												:= 'Reference rAxis invalid (0)';
	MemFnc													:= SEL(Execute , -1 ,MemFnc); 
	RETURN;
ELSIF NOT __ISVALIDREF(rMasterAxis)
THEN
	Busy													:= NOT Error;
	Error													:= TRUE;
	ErrorId													:= E_AdsErr.DEVICE_INVALIDPARM;
	CmdAborted												:= FALSE;
	Done													:= FALSE;
	ErrorText												:= 'Reference rMasterAxis invalid (0)';
	MemFnc													:= SEL(Execute , -1 ,MemFnc); 
	RETURN;
END_IF

	MC_GearInVelo(
		Execute			:= Execute,
		RatioNumerator	:= RatioNumerator ,
		RatioDenominator:= RatioDenominator ,
		SyncMode		:= SyncMode,
		Velocity		:= Velo,
		Acceleration	:= Acc,
		Deceleration	:= Dec,
		Jerk			:= Jerk,
		BufferMode		:= ,
		Options			:= ,
		Master			:= rMasterAxis,
		Slave			:= rAxis,
		StartSync		=> StartSync,
		InSync			=> Done,
		Busy			=> Busy,
		Active			=> Active,
		CommandAborted	=> CmdAborted,
		Error			=> Error,
		ErrorID			=> ErrorId);
	
	IF Error THEN
		LastErrorId											:= ErrorId;
		ErrorText 											:= CONCAT('MC_GearInVelo ID:' , UDINT_TO_STRING(ErrorId));
	ELSE
		ErrorText 											:= '';
	END_IF

	IF NOT Execute AND NOT Busy
	THEN
		MemFnc												:= -1;
	END_IF
	
	GearInVelo												:= Busy;
END_METHOD

METHOD PUBLIC gearOut : BOOL //Return value = TRUE if busy
//required parameter
//rAxis
VAR_INPUT
	Execute													:	BOOL;
END_VAR
MemFnc														:= FNC_GEAR_OUT;
THIS^.Execute												:= Execute;

IF NOT __ISVALIDREF(rAxis) 
THEN
	Busy													:= NOT Error;
	Error													:= TRUE;
	ErrorId													:= E_AdsErr.DEVICE_INVALIDPARM;
	CmdAborted												:= FALSE;
	Done													:= FALSE;
	Active													:= FALSE;
	ErrorText												:= 'Reference rAxis invalid (0)';
	MemFnc													:= SEL(Execute , -1 ,MemFnc); 
	RETURN;
END_IF

	MC_GearOut(
		Execute	:= Execute,
		Options	:= ,
		Slave	:= rAxis,
		Done	=> Done,
		Busy	=> Busy,
		Error	=> Error,
		ErrorID	=> ErrorID);

	Active													:= Busy;
	CmdAborted												:= FALSE;
	StartSync												:= FALSE;
	
	IF Error THEN
		LastErrorId											:= ErrorId;
		ErrorText 											:= CONCAT('MC_GearOut ID:' , UDINT_TO_STRING(ErrorId));
	ELSE
		ErrorText 											:= '';
	END_IF

	IF NOT Execute AND NOT Busy
	THEN
		MemFnc												:= -1;
	END_IF                  								
                            	
	GearOut													:= Busy;
END_METHOD

END_FUNCTION_BLOCK

// POUs/Motion/TF50xx-NC/02_Options/Coupling/AxGear
{attribute 'no_check'}
//Nc-axis gearing control 
//based on Tc2_MC2 library
FUNCTION_BLOCK AxGear EXTENDS AxFbBase
VAR_OUTPUT CONSTANT
	FNC_GEAR_OUT											:	INT := 0;
	FNC_GEAR_IN												:	INT := 1;
	FNC_GEAR_IN_DYN											:	INT := 2;
	FNC_GEAR_IN_MM											:	INT := 3;
END_VAR                     								
VAR_INPUT                   								
	Fnc														:	INT (FNC_GEAR_OUT..FNC_GEAR_IN_MM) := FNC_GEAR_OUT;
	RatioNumerator											:	LREAL := 1.0; // gear factor numerator
	RatioDenominator										:	UINT := 1; 	// gear factor denominator
	Acc														:	LREAL := 0.0; // if Acc = 0, the NC-Value will be set                         								
	Dec														:	LREAL := 0.0; // if Dec = 0, the NC-Value will be set
	Jerk													:	LREAL := 0.0; // if Jerk = 0, the NC-Value will be set
(*	
	BufferMode												:	MC_BufferMode := MC_Aborting;(* 	MC_Aborting,
																									MC_Buffered,
																									MC_BlendingLow,
																									MC_BlendingPrevious,
																									MC_BlendingNext,
																									MC_BlendingHigh *)
                            								
*)                          								
	OptionsGearInDyn										: 	ST_GearInDynOptions;
	OptionsGearInMM 										: 	ST_GearInMultiMasterOptions;
	
	rMasterAxis1											:	REFERENCE TO AXIS_REF := 0;
	rMasterAxis2											:	REFERENCE TO AXIS_REF := 0;
	rMasterAxis3											:	REFERENCE TO AXIS_REF := 0;
	rMasterAxis4											:	REFERENCE TO AXIS_REF := 0;
	MasterGearRatio1										:	LREAL := 1.0;
	MasterGearRatio2										:	LREAL := 1.0;
	MasterGearRatio3										:	LREAL := 1.0;
	MasterGearRatio4										:	LREAL := 1.0;
END_VAR                     								
VAR_IN_OUT                  								
END_VAR                     									
VAR_OUTPUT                  	
END_VAR
VAR
(* Zwischenspeicher **************************************************************************)
	MemFnc													:	INT := -1;

(* Trigger *)

(* Instanzierung der MC Bausteine *******************************************************)
	MC_GearInDyn											:	MC_GearInDyn;
	MC_GearIn												:	MC_GearIn;
	MC_GearOut												:	MC_GearOut;
	MC_GearInMultiMaster									:	MC_GearInMultiMaster;

(* Dummy Speicher **********************************************************)
(*	i,j		: INT := 0 ; *)
	Dummy 													: BOOL; 
END_VAR

	(************************************************************************************)
	(*																					*)
	(*		B E C K H O F F   N E W   A U T O M A T I O N   T E C H N O L O G Y    		*)
	(*																					*)
	(*		Eiserstr.5	D-33415 Verl	Germany	phone:	+49-5246-0	www.Beckhoff.Com	*)
    (*																					*)
    (*		Bausteinbeschreibung	:	Gear axis function-block						*)
	(*		TwinCAT-Version			:	3.x or higher		 							*)
	(*		Version					:	V3.1 / 01/14									*)
 	(*		Autor					:	Daniel Schlingmann								*)
	(*																					*)
	(************************************************************************************)

(* Execute ***************************************************************************************)
	rtExecute(CLK := Execute);
	IF rtExecute.Q
		AND MemFnc < 0
	THEN
		MemFnc 												:= Fnc ;
		Busy												:= TRUE;
		Done												:= FALSE;
		Active												:= FALSE;
		Error												:= FALSE;
		ErrorID												:= 0;
		CmdAborted											:= FALSE;
		ErrorText											:= '';
	END_IF

(* Call Method ***********************************************************************************)
	CASE MemFnc OF
	FNC_GEAR_OUT:
		GearOut(Execute);

	FNC_GEAR_IN:
		GearIn(Execute);

	FNC_GEAR_IN_DYN:
		GearInDyn(Execute);

	FNC_GEAR_IN_MM:
		GearInMM(Execute);

	-1:
		IF NOT Execute
		THEN
			Busy											:= FALSE;
			Done											:= FALSE;
			Active											:= FALSE;
			Error											:= FALSE;
			ErrorID											:= 0;
			CmdAborted										:= FALSE;
			ErrorText										:= '';
		END_IF                              				
	ELSE                                    				
		Busy												:= FALSE;
		Done												:= FALSE;
		Active												:= FALSE;
		Error												:= Execute;
		ErrorID												:= E_AdsErr.DEVICE_INVALIDPARM;
		CmdAborted											:= FALSE;
		ErrorText											:= CONCAT('invalid parameter value(s) Fnc no: ' , INT_TO_STRING(MemFnc));
	END_CASE                            		
                                            	

(*************************************************************************************************)

METHOD PUBLIC gearIn : BOOL //Return value = TRUE if busy
//required parameter
//rAxis
//rMasterAxis1
//RatioNumerator
//RatioDenominator
//Acc
VAR_INPUT
	Execute													:	BOOL;
END_VAR
MemFnc 														:= FNC_GEAR_IN;
THIS^.Execute												:= Execute;

IF NOT __ISVALIDREF(rAxis) 
THEN
	Busy													:= NOT Error;
	Error													:= TRUE;
	ErrorId													:= E_AdsErr.DEVICE_INVALIDPARM;
	CmdAborted												:= FALSE;
	Done													:= FALSE;
	Active													:= FALSE;
	ErrorText												:= 'Reference rAxis invalid (0)';
	MemFnc													:= SEL(Execute , -1 ,MemFnc); 
	RETURN;
ELSIF NOT __ISVALIDREF(rMasterAxis1)
THEN
	Busy													:= NOT Error;
	Error													:= TRUE;
	ErrorId													:= E_AdsErr.DEVICE_INVALIDPARM;
	CmdAborted												:= FALSE;
	Done													:= FALSE;
	ErrorText												:= 'Reference rMasterAxis1 invalid (0)';
	MemFnc													:= SEL(Execute , -1 ,MemFnc); 
	RETURN;
END_IF

	MC_GearIn(
		Execute				:= Execute,
		RatioNumerator		:= RatioNumerator,
		RatioDenominator	:= RatioDenominator,
		Acceleration		:= Acc,
		Deceleration		:= Dec,
		Jerk				:= Jerk,
		BufferMode			:= ,
		Options				:= ,
		Master				:= rMasterAxis1,
		Slave				:= rAxis,
		InGear				=> Done,
		Busy				=> Busy,
		Active				=> Active,
		CommandAborted		=> CmdAborted,
		Error				=> Error,
		ErrorID				=> ErrorID);

	IF Error THEN
		LastErrorId											:= ErrorId;
		ErrorText 											:= CONCAT('Error MC_GearIn ID:' , UDINT_TO_STRING(ErrorId));
	ELSE
		ErrorText 											:= '';
	END_IF

	IF NOT Execute AND NOT Busy
	THEN
		MemFnc												:=  -1;
	END_IF
	
	GearIn													:= Busy;
END_METHOD

METHOD PUBLIC gearInDyn : BOOL //Return value = TRUE if busy
//required parameter
//rAxis
//rMasterAxis1
//MasterGearRatio1
//Acc
VAR_INPUT
	Execute													:	BOOL;
END_VAR
MemFnc 														:= FNC_GEAR_IN_DYN;
THIS^.Execute												:= Execute;

IF NOT __ISVALIDREF(rAxis) 
THEN
	Busy													:= NOT Error;
	Error													:= TRUE;
	ErrorId													:= E_AdsErr.DEVICE_INVALIDPARM;
	CmdAborted												:= FALSE;
	Done													:= FALSE;
	Active													:= FALSE;
	ErrorText												:= 'Reference rAxis invalid (0)';
	MemFnc													:= SEL(Execute , -1 ,MemFnc); 
	RETURN;
ELSIF NOT __ISVALIDREF(rMasterAxis1)
THEN
	Busy													:= NOT Error;
	Error													:= TRUE;
	ErrorId													:= E_AdsErr.DEVICE_INVALIDPARM;
	CmdAborted												:= FALSE;
	Done													:= FALSE;
	ErrorText												:= 'Reference rMasterAxis1 invalid (0)';
	MemFnc													:= SEL(Execute , -1 ,MemFnc); 
	RETURN;
END_IF
	Dummy													:= MC_GearInDyn.Busy;
	MC_GearInDyn(
		Enable			:= Execute,
		GearRatio		:= MasterGearRatio1,
		Acceleration	:= Acc,
		Deceleration	:= Dec,
		Jerk			:= Jerk,
		BufferMode		:= ,
		Options			:= OptionsGearInDyn,
		Master			:= rMasterAxis1,
		Slave			:= rAxis,
		InGear			=> Done,
		Busy			=> Busy,
		Active			=> Active,
		CommandAborted	=> ,
		Error			=> ,
		ErrorID			=> );			

	IF NOT Busy AND(Dummy OR MC_GearInDyn.Enable)
	THEN
		CmdAborted											:= MC_GearInDyn.CommandAborted;
		Error												:=	MC_GearInDyn.Error;
		ErrorId												:= MC_GearInDyn.ErrorId;
		IF Error THEN           							
			LastErrorId											:= ErrorId;
			ErrorText 										:= CONCAT('MC_GearInDyn ID:' , UDINT_TO_STRING(ErrorId));
		ELSE                    							
			ErrorText 										:= '';
		END_IF                                          	
		IF NOT MC_GearInDyn.Enable                      	
		THEN                                            	
			MemFnc											:= -1;
		END_IF                                          	
	ELSE                                                	
		CmdAborted											:= FALSE;
		Error												:=	FALSE;
		ErrorId												:= 0;
		ErrorText 											:= '';
	END_IF                      							
	                            	                    	
	GearInDyn												:= Busy;
END_METHOD

METHOD PUBLIC gearInMM : BOOL//Return value = TRUE if busy
//required parameter
//rAxis
//rMasterAxis1
//rMasterAxis2
//rMasterAxis3
//rMasterAxis4
//MasterGearRatio1
//MasterGearRatio2
//MasterGearRatio3
//MasterGearRatio4
//Acc
VAR_INPUT
	Execute													:	BOOL;
END_VAR
MemFnc														:= FNC_GEAR_IN_MM;
THIS^.Execute												:= Execute;
	                										
IF NOT __ISVALIDREF(rAxis) 
THEN
	Busy													:= NOT Error;
	Error													:= TRUE;
	ErrorId													:= E_AdsErr.DEVICE_INVALIDPARM;
	CmdAborted												:= FALSE;
	Done													:= FALSE;
	Active													:= FALSE;
	ErrorText												:= 'Reference rAxis invalid (0)';
	MemFnc													:= SEL(Execute , -1 ,MemFnc); 
	RETURN;
ELSIF NOT __ISVALIDREF(rMasterAxis1)
	OR NOT __ISVALIDREF(rMasterAxis2)
	OR NOT __ISVALIDREF(rMasterAxis3)
	OR NOT __ISVALIDREF(rMasterAxis4) 
THEN
	Busy													:= NOT Error;
	Error													:= TRUE;
	ErrorId													:= E_AdsErr.DEVICE_INVALIDPARM;
	CmdAborted												:= FALSE;
	Done													:= FALSE;
	ErrorText												:= 'Reference rMasterAxis1..4 invalid (0)';
	MemFnc													:= SEL(Execute , -1 ,MemFnc); 
	RETURN;	
END_IF
	
	Dummy													:= MC_GearInMultiMaster.Busy;

	MC_GearInMultiMaster(
		Enable			:= Execute,
		GearRatio1		:= MasterGearRatio1,
		GearRatio2		:= MasterGearRatio2,
		GearRatio3		:= MasterGearRatio3,
		GearRatio4		:= MasterGearRatio4,
		Acceleration	:= Acc,
		Deceleration	:= Dec,
		Jerk			:= Jerk,
		BufferMode		:= ,
		Options			:= OptionsGearInMM,
		Master1			:= rMasterAxis1,
		Master2			:= rMasterAxis2,
		Master3			:= rMasterAxis3,
		Master4			:= rMasterAxis4,
		Slave			:= rAxis,
		InGear			=> Done,
		Busy			=> Busy,
		Active			=> Active,
		CommandAborted	=> ,
		Error			=> ,
		ErrorID			=> );							

	IF NOT Busy AND(Dummy OR MC_GearInMultiMaster.Enable)
	THEN
		CmdAborted											:= MC_GearInMultiMaster.CommandAborted;
		Error												:=	MC_GearInMultiMaster.Error;
		ErrorId												:= MC_GearInMultiMaster.ErrorId;
		IF Error 
		THEN
			LastErrorId										:= ErrorId;
			ErrorText 										:= CONCAT('MC_GearInMM ID:' , UDINT_TO_STRING(ErrorId));
		ELSE
			ErrorText 										:= '';
		END_IF
		IF NOT MC_GearInMultiMaster.Enable
		THEN
			MemFnc											:=  -1 ;
		END_IF                  							
	ELSE                        							
		CmdAborted											:= FALSE;
		Error												:=	FALSE;
		ErrorId												:= 0;
		ErrorText 											:= '';
	END_IF                      	
	
	GearInMM												:= Busy;
END_METHOD

METHOD PUBLIC gearOut : BOOL//Return value = TRUE if busy
//required parameter
//rAxis
VAR_INPUT
	Execute													:	BOOL;
END_VAR
IF NOT __ISVALIDREF(rAxis) 
THEN
	Busy													:= NOT Error;
	Error													:= TRUE;
	ErrorId													:= E_AdsErr.DEVICE_INVALIDPARM;
	CmdAborted												:= FALSE;
	Done													:= FALSE;
	Active													:= FALSE;
	ErrorText												:= 'Reference rAxis invalid (0)';
	MemFnc													:= SEL(Execute , -1 ,MemFnc); 
	RETURN;
END_IF

	MemFnc													:= FNC_GEAR_OUT;
	THIS^.Execute											:= Execute;
	
	MC_GearOut(
		Execute	:= Execute,
		Options	:= ,
		Slave	:= rAxis,
		Done	=> Done,
		Busy	=> Busy,
		Error	=> Error,
		ErrorID	=> ErrorID);

	Active													:= Busy;
	CmdAborted												:= FALSE;

	IF Error THEN
		LastErrorId											:= ErrorId;
		ErrorText 											:= CONCAT('MC_GearOut ID:' , UDINT_TO_STRING(ErrorId));
	ELSE
		ErrorText 											:= '';
	END_IF

	IF NOT Execute AND NOT Busy
	THEN
		MemFnc												:=  -1;
	END_IF                  								
                            	
	GearOut													:= Busy;
END_METHOD

END_FUNCTION_BLOCK

// POUs/Motion/TF50xx-NC/02_Options/Error/AxEventHandling
{attribute 'no_check'}
//EventHandlingGrp10 instance use inside
FUNCTION_BLOCK AxEventHandling
VAR CONSTANT
END_VAR                     								
VAR_INPUT                   								
	Enable													:	BOOL := TRUE; (* Show alarm message, warnings or hint. always reported !!! *)
	ConfirmTrig												:	BOOL := FALSE;
	SourceId												:	UDINT := 101000; //TwinCat-NC axis default multisource Id + Ax id
	ErrorId													:	UDINT := 0;
	Name													:	STRING(30) := '';
	rAxis													:	REFERENCE TO AXIS_REF := 0;
END_VAR
VAR_OUTPUT
{attribute 'displaymode':='binary'}
	Status													:	DWORD;
	NoOfActiveEvents										:	INT;
END_VAR
VAR
(* Zwischenspeicher ***********************************************)
	QuitInternal 											: BOOL;

(* Timer **********************************************************)

(* Trigger ********************************************************)

(* Bausteine ******************************************************)
	Event													:	EventHandlingGrp10 := (
																	AutoConfirm			:= FALSE, 
																	SetClass 			:= TC2_SYSTEM.TCEVENTCLASS_ALARM );
	AxNcEvent												:	AxNcEventHandling;

(* Dummy Speicher *************************************************)
	i														:	INT ;

END_VAR

(* Error message axis to EventLogger 			V3.0	DS	*)
(***********************************************************)

(* Sequence **************************************************************)
IF __ISVALIDREF(rAxis) 
THEN
	(* get Quit signal **************************************************)
	IF ConfirmTrig 
	THEN 
		QuitInternal 										:= TRUE; 
	END_IF (* set false see below *)

(* Event Logger Meldungen *****************************************************)
	Event.no[1].Flag 										:= rAxis.Status.IoDataInvalid;
	Event.no[2].Flag 										:= rAxis.Status.DriveDeviceError;
	Event.no[3].Flag 										:= rAxis.Status.Homing;   
	Event.no[4].Flag 										:= rAxis.Status.SoftLimitMinExceeded AND rAxis.Status.Homed AND NOT rAxis.Status.InTargetPosition; //Show msg only if SW is reached without active movement   
	Event.no[5].Flag 										:= rAxis.Status.SoftLimitMaxExceeded AND rAxis.Status.Homed AND NOT rAxis.Status.InTargetPosition; 	//Show msg only if SW is reached without active movement   
(*
	Event.no[6].Flag 										:= FALSE;
	Event.no[7].Flag 										:= FALSE;
	Event.no[8].Flag 										:= FALSE;
	Event.no[9].Flag 										:= FALSE;
	Event.no[10].Flag 										:= FALSE;
*)
(* workl Event Ctrl *************************************************)
	IF Event.no[1].Text2 <> Name AND Name <> '' OR Event.no[1].Text2 = '' AND AxisId <> 0
	THEN
		//Init EventClass
		Event.no[3].eClass 									:= TC2_SYSTEM.TCEVENTCLASS_HINT;
		Event.no[4].eClass 									:= TC2_SYSTEM.TCEVENTCLASS_STATEINFO;
		Event.no[5].eClass 									:= TC2_SYSTEM.TCEVENTCLASS_STATEINFO;

		(* Init Name *)
		FOR i := Event.MIN_EVENT TO Event.MAX_EVENT DO
			Event.no[i].Text2								:= SEL(LEN(name)>1,CONCAT('Axis id:',DWORD_TO_STRING(rAxis.NcToPlc.AxisId)),name);
		END_FOR
	END_IF

	Event(
		ConfirmTrig := ConfirmTrig,
		Disable		:= NOT Enable,
		SourceId	:= SourceId + rAxis.NcToPlc.AxisId,
		Status	 	=> );	

(* Send ErrorId Message Text **********************************)
	AxNcEvent(
		ConfirmTrig	:= NOT Enable OR QuitInternal OR ErrorId = 0 AND AxNcEvent.State <> 0,
		Name		:= name,
		AxisId		:= rAxis.NcToPlc.AxisId,
		SourceId	:= SourceId,
		Flag		:= ErrorId > 0 AND Enable,
		ErrorID		:= ErrorId,
		State		=> );

(* EventStatus *************************************************)
	Status													:= AxNcEvent.Status OR Event.Status;
	NoOfActiveEvents										:= Event.NoOfActiveEvents + SEL(AxNcEvent.Status.31 , 0, 1);

(* Error unkonw pointer or axis id *****************************)
ELSE
	NoOfActiveEvents										:= 0;
	AxNcEvent(Flag := FALSE, ConfirmTrig := AxNcEvent.State <> 0);
	Event(Disable := TRUE, Status =>  ); 
	Status													:= AxNcEvent.Status OR Event.Status;
END_IF

(* Default reset Quit Internal *******************************)
	QuitInternal 											:= FALSE;

(**************************************************************)

METHOD PUBLIC confirm : bool //Return value = TRUE if execution finished 
VAR_INPUT
END_VAR
QuitInternal 												:= TRUE;
confirm													:= TRUE;
END_METHOD

END_FUNCTION_BLOCK

// POUs/Motion/TF50xx-NC/02_Options/Error/AxNcEventHandling
{attribute 'no_check'}
FUNCTION_BLOCK AxNcEventHandling
VAR CONSTANT
END_VAR     
VAR_INPUT
	Flag													:	BOOL := FALSE;  
	ConfirmTrig													:	BOOL := FALSE;
	MsgId													:	UDINT := 201; //Default
	SourceId												:	UDINT := 101000; //TwinCat-NC axis default multisource Id + Ax id for detailed event message
	AxisId													:	UDINT := 0;
	ErrorID													:	UDINT := 0; (* NC Error Id Bsp 18000 -Drive Error *)
	Name													: 	STRING(30) := '';
END_VAR                         							
VAR_OUTPUT                      							
	State													:	UDINT := TCEVENTSTATE_INVALID;
																		(* TCEVENTSTATE_INVALID  	: WORD := 16#0000; (* Ungültig, kommt auch wenn Event noch nicht gemeldet. *)
																			TCEVENTSTATE_SIGNALED  	: WORD := 16#0001; (* Event ist gemeldet, aber weder gegangen noch quittiert. *)
																			TCEVENTSTATE_RESET  		: WORD := 16#0002; (* Event ist abgemeldet ('gegangen'). *)
																			TCEVENTSTATE_CONFIRMED  : WORD := 16#0010 (16); (* Event ist quittiert. *)
																			TCEVENTSTATE_RESETCON  	: WORD := 16#0012 (17); (* Event ist abgemeldet und quittiert *) *)
{attribute 'displaymode':='binary'}
	Status													:	DWORD; (*	.0 - .8 = event <class id>  / .15 Quit required / .16 = Level 0 , .17 = Level 1 , .18 = Level 2, .......... / .31 active
																			TCEVENTCLASS_NONE			:=0,	(* No class *)
																			TCEVENTCLASS_MAINTENANCE	:=1,	(* Maintenance hint *)
																			TCEVENTCLASS_MESSAGE		:=2,	(* Message *)
																			TCEVENTCLASS_HINT			:=3,	(* Hint *)
																			TCEVENTCLASS_STATEINFO		:=4,	(* State information *)
																			TCEVENTCLASS_INSTRUCTION	:=5,	(* Instruction *)
																			TCEVENTCLASS_WARNING		:=6,	(* Warning *)
																			TCEVENTCLASS_ALARM			:=7,	(* Alarm *)
																			TCEVENTCLASS_PARAMERROR		:=8		(* Parameter error *)  *)
END_VAR
VAR
	AdsEvent												:		ADSLOGEVENT :=(
																		Event			:= FALSE,
																		NETID			:= '',
																		PORT			:= AMSPORT_EVENTLOG,
																		TMOUT 			:= DEFAULT_ADS_TIMEOUT,
																		EventConfigData := (
																					Class 			:= TC2_SYSTEM.TCEVENTCLASS_ALARM,
																					Prio 			:= TCEVENTPRIO_IMPLICIT,
																					ProgId 			:= 'TcEventFormatter.TcXmlFormatter',
																					Flags 			:= 16#0140 (* TCEVENTFLAG_LOG OR TCEVENTFLAG_SRCID *),
																					StreamType 		:= TCEVENTSTREAM_NORMAL (* TCEVENTSTREAM_SIMPLE *),
																					bQuitRequired 	:= FALSE));
                    										
	FormatString 											: STRING(15) := '%s%d%s%s%d%s';
                    										
	pParaArray												: ARRAY [1..6] OF PVOID;
                    										
	Para1													: STRING(30);
	Para2													: UDINT;
	Para3													: STRING(70);
	Para4													: STRING(70);
	Para5													: UDINT;
	Para6													: STRING(20);
	SetClass												: E_TcEventClass := TC2_SYSTEM.TCEVENTCLASS_ALARM;
END_VAR

(* Send axis error text to EventLogger		 							*)
(************************************************************************)

(* Event Config ************************************************)
	IF Status.31 //Message active
	THEN (* work EventLogger *)

		AdsEvent(
			NETID			:= ,(* siehe deklaration *)
			PORT			:= ,(* siehe deklaration *)
			Event			:= NOT AdsEvent.FbCleanup AND(Flag AND Para2 = ErrorID OR AdsEvent.EventState = TCEVENTSTATE_INVALID AND NOT AdsEvent.Quit),
			EventQuit		:= AdsEvent.EventState <> TCEVENTSTATE_INVALID
								AND AdsEvent.EventConfigData.bQuitRequired
								AND NOT AdsEvent.Eventstate.4
								AND NOT AdsEvent.Quit
								AND(
								ConfirmTrig
								OR Para2 <> ErrorID
								OR AdsEvent.EventQuit), (* quit send *)
			EventConfigData	:= ,(* siehe deklaration *)
			EventDataAddress:= ADR(pParaArray),
			EventDataLength	:= ,
			FbCleanup		:= NOT AdsEvent.FbCleanup AND(AdsEvent.Err OR AdsEvent.EventState = TCEVENTSTATE_RESETCON),
			TMOUT			:= ,(* siehe deklaration *)
			EventState		=> ,
			Err				=> ,
			ErrId			=> ,
			Quit			=> );

		IF AdsEvent.Event
			AND AdsEvent.EventState = TCEVENTSTATE_INVALID
		THEN
			State 											:= SEL(Flag, TCEVENTSTATE_RESET, TCEVENTSTATE_SIGNALED);
		ELSIF AdsEvent.Quit
			AND AdsEvent.EventState = TCEVENTSTATE_INVALID
			AND AdsEvent.EventQuit
			OR 
			AdsEvent.FbCleanup		
		THEN
			State 											:= TCEVENTSTATE_RESETCON;
		ELSIF(AdsEvent.Err OR NOT AdsEvent.Event AND AdsEvent.EventState = TCEVENTSTATE_INVALID)
			AND_THEN Gvl.EventHandlingStatistic.CountOut(Status)
		THEN
			State											:= TCEVENTSTATE_INVALID;
		ELSE
			State											:= MAX(State, AdsEvent.EventState);
		END_IF
	
	ELSIF flag AND SourceId > 0
	THEN (* fire event *)
	(*	Type : 2 - Axis Event 201
		%1 User Name 
		%2 	Unique error id (DINT)
		%3	Error text (STRING) ) Bsp.: [S750E20392]
		@V1:%4	Error description (STRING) Bsp.: [S751E20392]
		%5	Logical axis id (DINT)
		@V2:%6	Position OF axis (REAL) or Reserved text 
	
	*)
		Para1 												:= Name;
		Para2 												:= ErrorID;
              												
		Para3 												:= CONCAT('[S','700'); (* SOURCE_TEXT_PTPNCI = 701 *)
		Para3 												:= CONCAT(Para3,'E');
		Para3 												:= CONCAT(Para3,UDINT_TO_STRING(ErrorID));
		Para3 												:= CONCAT(Para3,']');
              												
		Para4 												:= CONCAT('[S','701'); (* SOURCE_DESC_PTPNCI = 701 *)
		Para4 												:= CONCAT(Para4,'E');
		Para4 												:= CONCAT(Para4,UDINT_TO_STRING(ErrorID));
		Para4 												:= CONCAT(Para4,']');
              												
		Para5 												:= AxisId;
		Para6 												:= ''; (* Reserve *)

		pParaArray[1] 										:= ADR(Para1);
		pParaArray[2] 										:= ADR(Para2);
		pParaArray[3] 										:= ADR(Para3);
		pParaArray[4] 										:= ADR(Para4);
		pParaArray[5] 										:= ADR(Para5);
		pParaArray[6] 										:= ADR(Para6);

		
		AdsEvent.EventConfigData.Id 						:= MsgId; (* MSG_ID = 201 *)
 		AdsEvent.EventConfigData.DataFormatStrAddress 		:= ADR(FormatString);
		AdsEvent.EventConfigData.SourceId 					:= SourceId + AxisId;
		Status												:= Gvl.EventHandlingStatistic.InitEvent(SetClass , AdsEvent.EventConfigData);	

		IF AdsEvent.Err AND NOT AdsEvent.FbCleanup
		THEN
			AdsEvent(
				Event			:= FALSE,
				EventQuit 		:= FALSE,
				EventDataAddress:= ADR(pParaArray),
				FbCleanup		:= TRUE,
				EventState		=> );
		
		ELSE (* Fire Event *)
			AdsEvent( 	Event			:= FALSE,
						EventQuit 		:= FALSE, 
						FbCleanup 		:= FALSE, 
						EventDataAddress:= ADR(pParaArray));
			AdsEvent( 	Event 	:= TRUE);			
			IF NOT AdsEvent.Err AND_THEN Gvl.EventHandlingStatistic.CountIn(Status) //Add event to statistic and continue if added successfully
			THEN			
				State 										:= TCEVENTSTATE_SIGNALED;
			END_IF
		END_IF
	END_IF

(*****************************************************************)

END_FUNCTION_BLOCK

// POUs/Motion/TF50xx-NC/02_Options/Motion/AxHomingOnBlock
{attribute 'no_check'}
//Nc-axis homing on block sequence control for CoE drive 
//based on Tc2_MC2 library
FUNCTION_BLOCK AxHomingOnBlock EXTENDS FbBase
VAR CONSTANT	
	DEVICE_TYPE_PROFILE_DS402								:	UDINT := 5001;
	DEVICE_TYPE_PROFILE_MDP									:	UDINT := 131474;	
END_VAR
VAR_INPUT
	Position												: LREAL := DEFAULT_HOME_POSITION;//Used as homepos if value is <> DEFAULT_HOME_POSITION
	Direction												: MC_Direction := MC_Negative_Direction; //Homing direction
	Velocity												: LREAL := 0.0; //0.0 = Default NC valuse are used, else "Velocity" is used for both movements, into block direction and retraction
	Acceleration											: LREAL := 0.0; //0.0 = Default dynamics are used
	Deceleration											: LREAL := 0.0; //0.0 = Default dynamics are used
	Offset													: LREAL := 2.0; //Offset to release block
	LagTolerance											: LREAL	:= 0.5; //Lag error tolerance to detect axis on block
	MaxTorque												: LREAL	:= 50.0;//Max torque during homing towards block and retartion
	DrvChannel												: BYTE	:= 0; //Drive channel 0 or 1 
END_VAR
VAR_IN_OUT
	Axis													: AXIS_REF;
END_VAR
VAR_OUTPUT
	DriveProfileIsDS402										:	BOOL;							
END_VAR
VAR
(* Internal memory **********************************************************************)
	LastErrorState											: INT ; //Last error state for debugging
	LastErrorId												: UDINT;
	MemError												: BOOL;
	MemBlockPos												: LREAL;
	VelocityTowardsBlock									: LREAL;
	VelocityOffBlock										: LREAL;
	// Parameter storage for returning values to original after running the procedure.
	Param_DeviceType										: UDINT;
	Param_MotionMonitoring									: BYTE;
	Param_LagMonitoring										: BYTE;
	Param_SoftMaxMonitoring									: BYTE;
	Param_SoftMinMonitoring									: BYTE;	                        	
	Param_MaxTorque											: UINT;
	Param_MaxTorqueRead										: BOOL;
	Param_CalibrationValue									: LREAL;
	
(* Timer ********************************************************************************)                 	

(* Trigger ******************************************************************************)

(* FB instances *************************************************************************)
	Read_ADS												: ADSREAD := (TmOut := DEFAULT_ADS_TIMEOUT);
	Write_ADS												: ADSWRITE  := (TmOut := DEFAULT_ADS_TIMEOUT);
	MC_Home													: MC_Home;
	Mc_Halt													: MC_Halt;
	MC_Velocity												: MC_MoveVelocity;
	MC_Absolute												: MC_MoveAbsolute;
	CoEWrite												: FB_CoEWrite;
	CoERead													: FB_CoERead;
(* Dummys *******************************************************************************)
	uiValue													: UINT; //Temporary use for reading BOOL
END_VAR

	(* Homing on block function																		*)
	(*																								*)
	(* V1.0 2016/02/15 ABarrett																		*)
	(************************************************************************************************)
	
(* Sequence *************************************************************************************)
rtExecute(CLK := Execute);
CASE State OF
0://Wait for execute signal to change state to true
	IF NOT Execute OR rtExecute.Q	
	THEN
		Read_ADS(Read := FALSE);	Write_Ads(Write := FALSE);
		CoEWrite(Execute := FALSE,axis  := axis); CoERead(Execute := FALSE,axis  := axis);										
		MC_Home(Execute := FALSE,Axis := Axis);
		MC_Halt(Execute := FALSE,Axis := Axis);
		MC_Velocity(Execute := FALSE,Axis := Axis);
		MC_Absolute(Execute := FALSE,Axis := Axis);	
		Param_MotionMonitoring								:= 0;
		Param_LagMonitoring									:= 0;
		Param_SoftMaxMonitoring								:= 0;
		Param_SoftMinMonitoring								:= 0;
	
		Busy												:= rtExecute.Q;
		Done 												:= FALSE;
		Error												:= FALSE;
		ErrorID												:= 0;
		MemError											:= 0;
		state												:= SEL(rtExecute.Q, 0, 100);
	
	END_IF

(* Read original parameters for position lag monitoring, limit switches, max torque....... ************************************)
100:
	(* Read device type from drive *)
	CoERead( 
		NetId			:= '', 
		Index			:= 16#1000,
		SubIndex		:= 0, 
		pDstBuf			:= ADR(Param_DeviceType), 
		BufLen			:= SIZEOF(Param_DeviceType), 
		Execute			:= TRUE, 
		Axis			:= Axis );
	IF NOT CoERead.BUSY
	THEN
		IF CoERead.Error
		THEN
			MemError										:= TRUE;
			LastErrorState									:= state;
			LastErrorId										:= CoERead.AdsErrId;//or CANopenErrId;				
			State											:= 900;
		ELSE
			DriveProfileIsDS402								:= Param_DeviceType = DEVICE_TYPE_PROFILE_DS402; 
			CoERead(Execute := FALSE, Axis := Axis);	
			state											:= State + 1;
		END_IF		
	END_IF

101:
	Read_ADS(NetId:= '' , Port:=500, IdxGrp:=16#4000+Axis.NcToPlc.AxisId, IDxOffs:=16#11,
				LEN:=SIZEOF(uiValue), DestAddr:=ADR(uiValue), Read := TRUE );
	IF NOT Read_ADS.BUSY 
	THEN
		IF Read_Ads.ERR
		THEN
			MemError										:= TRUE;
			LastErrorState									:= state;
			LastErrorId										:= Read_Ads.ERRID;				
			State											:= 900;
		ELSE                                            	
			Param_MotionMonitoring.0						:= TRUE;                                    	
			Param_MotionMonitoring.1						:= TO_BOOL(uiValue);
			state											:= state + 1;
		END_IF
		Read_ADS(Read := FALSE);						
	END_IF
	
102:
	Read_ADS(NetId:= '' , Port:=500, IdxGrp:=16#6000+Axis.NcToPlc.AxisId, IDxOffs:=16#10,
				LEN:=SIZEOF(uiValue), DestAddr:=ADR(uiValue), Read := TRUE );
	IF NOT Read_ADS.BUSY 
	THEN
		IF Read_Ads.ERR
		THEN
			MemError										:= TRUE;
			LastErrorState									:= state;
			LastErrorId										:= Read_Ads.ERRID;				
			State											:= 900;
		ELSE                                            	
			Param_LagMonitoring.0							:= TRUE;                                    	
			Param_LagMonitoring.1							:= TO_BOOL(uiValue);
			state											:= state + 1;
		END_IF
		Read_ADS(Read := FALSE);						
	END_IF		
		
103:
	Read_ADS(NetId:= '' , Port:=500, IdxGrp:=16#5000+Axis.NcToPlc.AxisId, IDxOffs:=16#C,
				LEN:=SIZEOF(uiValue), DestAddr:=ADR(uiValue), Read := TRUE );
	IF NOT Read_ADS.BUSY 
	THEN
		IF Read_Ads.ERR
		THEN
			MemError										:= TRUE;
			LastErrorState									:= state;
			LastErrorId										:= Read_Ads.ERRID;				
			State											:= 900;
		ELSE                                            	
			Param_SoftMaxMonitoring.0						:= TRUE;                                    	
			Param_SoftMaxMonitoring.1						:= TO_BOOL(uiValue);
			state											:= state + 1;
		END_IF
		Read_ADS(Read := FALSE);						
	END_IF		
	
104:
	Read_ADS(NetId:= '' , Port:=500, IdxGrp:=16#5000+Axis.NcToPlc.AxisId, IDxOffs:=16#B,
				LEN:=SIZEOF(uiValue), DestAddr:=ADR(uiValue), Read := TRUE );
	IF NOT Read_ADS.BUSY 
	THEN
		IF Read_Ads.ERR
		THEN
			MemError										:= TRUE;
			LastErrorState									:= state;
			LastErrorId										:= Read_Ads.ERRID;				
			State											:= 900;
		ELSE                                            	
			Param_SoftMinMonitoring.0						:= TRUE;                                    	
			Param_SoftMinMonitoring.1						:= TO_BOOL(uiValue);
			state											:= State + 1;
		END_IF
		Read_ADS(Read := FALSE);						
	END_IF	

105:
	Read_ADS(NetId:= '' , Port:=500, IdxGrp:=16#5000+Axis.NcToPlc.AxisId, IDxOffs:=16#103,
				LEN:=SIZEOF(Param_CalibrationValue), DestAddr:=ADR(Param_CalibrationValue), Read := TRUE );
	IF NOT Read_ADS.BUSY 
	THEN
		IF Read_Ads.ERR
		THEN
			MemError										:= TRUE;
			LastErrorState									:= state;
			LastErrorId										:= Read_Ads.ERRID;				
			State											:= 900;
		ELSE                                            	
			state											:= State + 1;
		END_IF
		Read_ADS(Read := FALSE);						
	END_IF			
	
106://Read velocity to use towards block
	IF Velocity = 0.0
	THEN //Only read values if FB parameter is 0.0
		Read_ADS(NetId:= '' , Port:=500, IdxGrp:=16#4000+Axis.NcToPlc.AxisId, IDxOffs:=16#6,
					LEN:=SIZEOF(VelocityTowardsBlock), DestAddr:=ADR(VelocityTowardsBlock), Read := TRUE );
		IF NOT Read_ADS.BUSY 
		THEN
			IF Read_Ads.ERR
			THEN
				MemError									:= TRUE;
				LastErrorState								:= state;
				LastErrorId									:= Read_Ads.ERRID;				
				State										:= 900;
			ELSE                                            
				state										:= State + 1;
			END_IF                                          
			Read_ADS(Read := FALSE);						
		END_IF                                              
	ELSE	                                                
		VelocityTowardsBlock								:= Velocity;
		VelocityOffBlock									:= Velocity;
		state												:= 108;	//Skip this and next state
	END_IF
	
107://Read velocity to use away from block to home position
	Read_ADS(NetId:= '' , Port:=500, IdxGrp:=16#4000+Axis.NcToPlc.AxisId, IDxOffs:=16#7,
				LEN:=SIZEOF(VelocityOffBlock), DestAddr:=ADR(VelocityOffBlock), Read := TRUE );
	IF NOT Read_ADS.BUSY 
	THEN
		IF Read_Ads.ERR
		THEN
			MemError										:= TRUE;
			LastErrorState									:= state;
			LastErrorId										:= Read_Ads.ERRID;				
			State											:= 900;
		ELSE                                            	
			state											:= State + 1;
		END_IF
		Read_ADS(Read := FALSE);						
	END_IF	
		
108://Read CoE value for max torque
	IF DrvChannel = 1
	THEN
		CoERead.Index										:= SEL(DriveProfileIsDS402, 16#7110 , 	16#6872); 
		CoERead.SubIndex									:= SEL(DriveProfileIsDS402, 16#B  , 	16#0);
	ELSE //Channel 0
		CoERead.Index										:= SEL(DriveProfileIsDS402, 16#7010 , 	16#6072);
		CoERead.SubIndex									:= SEL(DriveProfileIsDS402, 16#B  , 	16#0);
 	END_IF 
	
	CoERead( 
		NetId			:= '', 
		Index			:= , //See above 
		SubIndex		:= , //See above 
		pDstBuf			:= ADR(uiValue), 
		BufLen			:= SIZEOF(uiValue), //2,
		Execute			:= TRUE, 
		Axis			:= Axis );
	IF NOT CoERead.BUSY
	THEN
		IF CoERead.Error
		THEN
			MemError										:= TRUE;
			LastErrorState									:= state;
			LastErrorId										:= CoERead.AdsErrId;//or CANopenErrId;				
			State											:= 900;
		ELSE
			Param_MaxTorqueRead								:= TRUE;
			Param_MaxTorque									:= uiValue;
			CoERead(Execute := FALSE, Axis := Axis);	
			state											:= 200;
		END_IF		
	END_IF
	
	
(* Write all parameters to needed settings *********************************************************)
200:
	uiValue													:= TO_UINT(FALSE);
	Write_ADS(NetId:= '' , Port:=500, IdxGrp:=16#4000+Axis.NcToPlc.AxisId, IDxOffs:=16#11,
				LEN:=SIZEOF(uiValue), SrcAddr:=ADR(uiValue), Write := TRUE );
	IF NOT Write_ADS.BUSY 
	THEN
		IF Write_ADS.ERR
		THEN
			MemError										:= TRUE;
			LastErrorState									:= state;
			LastErrorId										:= Read_Ads.ERRID;				
			State											:= 600; //Jump to state 600 to restore old entrys
		ELSE
			state											:= state + 1;
		END_IF
		Write_ADS(Write := FALSE);						
	END_IF

201:
	uiValue													:= TO_UINT(FALSE);
	Write_ADS(NetId:= '' , Port:=500, IdxGrp:=16#6000+Axis.NcToPlc.AxisId, IDxOffs:=16#10,
				LEN:=SIZEOF(uiValue), SrcAddr:=ADR(uiValue), Write := TRUE );
	IF NOT Write_ADS.BUSY 
	THEN
		IF Write_ADS.ERR
		THEN
			MemError										:= TRUE;
			LastErrorState									:= state;
			LastErrorId										:= Read_Ads.ERRID;				
			State											:= 600; //Jump to state 600 to restore old entrys
		ELSE
			state											:= state + 1;
		END_IF
		Write_ADS(Write := FALSE);						
	END_IF

202:	
	uiValue													:= TO_UINT(FALSE);
	Write_ADS(NetId:= '' , Port:=500, IdxGrp:=16#5000+Axis.NcToPlc.AxisId, IDxOffs:=16#C,
					LEN:=SIZEOF(uiValue), SrcAddr:=ADR(uiValue), Write := TRUE );
	IF NOT Write_ADS.BUSY 
	THEN
		IF Write_ADS.ERR
		THEN
			MemError										:= TRUE;
			LastErrorState									:= state;
			LastErrorId										:= Read_Ads.ERRID;				
			State											:= 600; //Jump to state 600 to restore old entrys
		ELSE
			state											:= state + 1;
		END_IF
		Write_ADS(Write := FALSE);						
	END_IF
	
203:	
	uiValue													:= TO_UINT(FALSE);
	Write_ADS(NetId:= '' , Port:=500, IdxGrp:=16#5000+Axis.NcToPlc.AxisId, IDxOffs:=16#B,
					LEN:=SIZEOF(uiValue), SrcAddr:=ADR(uiValue), Write := TRUE );
	IF NOT Write_ADS.BUSY 
	THEN
		IF Write_ADS.ERR
		THEN
			MemError										:= TRUE;
			LastErrorState									:= state;
			LastErrorId										:= Read_Ads.ERRID;				
			State											:= 600; //Jump to state 600 to restore old entrys
		ELSE
			state											:= 204;
		END_IF
		Write_ADS(Write := FALSE);						
	END_IF

	
204://Write the max torque value used for homing
	IF DrvChannel = 1
	THEN
		CoERead.Index										:= SEL(DriveProfileIsDS402, 16#7110 , 	16#6872); 
		CoERead.SubIndex									:= SEL(DriveProfileIsDS402, 16#B  , 	16#0);
	ELSE //Channel 0
		CoERead.Index										:= SEL(DriveProfileIsDS402, 16#7010 , 	16#6072);
		CoERead.SubIndex									:= SEL(DriveProfileIsDS402, 16#B  , 	16#0);
 	END_IF 

	uiValue													:= LREAL_TO_UINT(MaxTorque) * 10;
	CoEWrite(
		NetId			:= '', 
		Index			:= , //See above
		SubIndex		:= , //See above
		pSrcBuf			:= ADR(uiValue), 
		BufLen			:= SIZEOF(uiValue),//2, 
		Execute			:= TRUE, 
		Axis			:= Axis
	);
	IF NOT CoEWrite.BUSY 
	THEN
		IF CoEWrite.Error
		THEN
			MemError										:= TRUE;
			LastErrorState									:= state;
			LastErrorId										:= CoEWrite.AdsErrId;//or CANopenErrId;				
			State											:= 600; //Jump to state 600 to restore old entrys
		ELSE
			state											:= 300;
		END_IF
		CoEWrite(Execute := FALSE, Axis := Axis);						
	END_IF
	
(* Velocity move until Homing_Tolerance exceeded *****************************************************************)
300:
	MC_Velocity( 
		Axis			:= Axis,
		Execute			:= TRUE,
		Velocity		:= VelocityTowardsBlock,
		Direction		:= Direction,
		Acceleration	:= Acceleration,
		Deceleration	:= Deceleration
	);
	
	IF ABS(Axis.NcToPlc.PosDiff) > lagTolerance
		OR NOT MC_Velocity.Busy //In case and error occure, the state machine can still continie
	THEN
		IF MC_Velocity.Error
		THEN
			MemError										:= TRUE;
			LastErrorState									:= state;
			LastErrorId										:= MC_Velocity.ErrorID;	
			state											:= 600; //Try to restore old parameter first
		ELSE
			MemBlockPos										:= Axis.NcToPlc.ActPos; //Record block pos
			MC_Halt(Execute := TRUE, Axis := Axis);
			State 											:= state + 1;
		END_IF
		MC_Velocity(Execute := FALSE, Axis := Axis);
	END_IF
	
301: //Wait for movment stopped 
	MC_Halt(Execute := TRUE, Axis := Axis);
	IF NOT MC_Halt.Busy
	THEN
		IF MC_Halt.Error
		THEN
			MemError										:= TRUE;
			LastErrorState									:= state;
			LastErrorId										:= MC_Halt.ErrorID;	
			state											:= 600; //Try to restore old parameter first		
		ELSE	
			state											:= 400; 	
		END_IF
		MC_Halt(Execute := FALSE, Axis := Axis);
	END_IF
	
400://Move to offset 
	MC_Absolute(
		Axis			:= Axis,
		Execute			:= TRUE,		
		Position		:= MemBlockPos + (ABS(Offset) * SEL(MC_Velocity.Direction = MC_Negative_Direction, -1.0 , 1.0)), //Calculate offset direction automaically 
		Velocity		:= VelocityOffBlock,
		Acceleration	:= Acceleration,
		Deceleration	:= Deceleration
	);
	IF NOT MC_Absolute.Busy 
	THEN
		IF MC_Absolute.Error
		THEN
			MemError										:= TRUE;
			LastErrorState									:= state;
			LastErrorId										:= MC_Absolute.ErrorID;	
			state											:= 600; //Try to restore old parameter first		
		ELSE	
			state											:= 500; 	
		END_IF
		MC_Absolute(Execute := FALSE, Axis := Axis);
	END_IF
	
